   1:  PR[GP1:91,2] = PR[GP1:90,2] + 0.302;
   1:L PR[91] 10mm/sec CNT100;
   1:  PR[GP1:91,1] = PR[GP1:90,1] + 73.416;
   1:  PR[GP1:91,2] = PR[GP1:90,2] + 5.594;
   1:L PR[91] 10mm/sec CNT100;
   1:  PR[GP1:91,1] = PR[GP1:90,1] + 72.687;
   1:  PR[GP1:91,2] = PR[GP1:90,2] + 9.406;
   1:L PR[91] 10mm/sec CNT100;
   1:  PR[GP1:91,1] = PR[GP1:90,1] + 70.980;
   1:  PR[GP1:91,2] = PR[GP1:90,2] + 14.355;
   1:L PR[91] 10mm/sec CNT100;
   1:  PR[GP1:91,1] = PR[GP1:90,1] + 68.206;
   1:  PR[GP1:91,2] = PR[GP1:90,2] + 18.843;
   1:L PR[91] 10mm/sec CNT100;
   1:  PR[GP1:91,1] = PR[GP1:90,1] + 66.056;
   1:  PR[GP1:91,2] = PR[GP1:90,2] + 22.237;
   1:L PR[91] 10mm/sec CNT100;
   1:  PR[GP1:91,1] = PR[GP1:90,1] + 62.477;
   1:  PR[GP1:91,2] = PR[GP1:90,2] + 25.890;
   1:L PR[91] 10mm/sec CNT100;
   1:  PR[GP1:91,1] = PR[GP1:90,1] + 58.115;
   1:  PR[GP1:91,2] = PR[GP1:90,2] + 28.712;
   1:L PR[91] 10mm/sec CNT100;
   1:  PR[GP1:91,1] = PR[GP1:90,1] + 54.751;
   1:  PR[GP1:91,2] = PR[GP1:90,2] + 31.172;
   1:L PR[91] 10mm/sec CNT100;
   1:  PR[GP1:91,1] = PR[GP1:90,1] + 50.096;
   1:  PR[GP1:91,2] = PR[GP1:90,2] + 32.886;
   1:L PR[91] 10mm/sec CNT100;
   1:  PR[GP1:91,1] = PR[GP1:90,1] + 45.611;
   1:  PR[GP1:91,2] = PR[GP1:90,2] + 34.049;
   1:L PR[91] 10mm/sec CNT100;
   1:  PR[GP1:91,1] = PR[GP1:90,1] + 40.919;
   1:  PR[GP1:91,2] = PR[GP1:90,2] + 34.669;
   1:L PR[91] 10mm/sec CNT100;
   1:  PR[GP1:91,1] = PR[GP1:90,1] + 36.178;
   1:  PR[GP1:91,2] = PR[GP1:90,2] + 34.240;
   1:L PR[91] 10mm/sec CNT100;
   1:  PR[GP1:91,1] = PR[GP1:90,1] + 31.221;
   1:  PR[GP1:91,2] = PR[GP1:90,2] + 33.641;
   1:L PR[91] 10mm/sec CNT100;
   1:  PR[GP1:91,1] = PR[GP1:90,1] + 27.016;
   1:  PR[GP1:91,2] = PR[GP1:90,2] + 32.287;
   1:L PR[91] 10mm/sec CNT100;
   1:  PR[GP1:91,1] = PR[GP1:90,1] + 23.151;
   1:  PR[GP1:91,2] = PR[GP1:90,2] + 30.007;
   1:L PR[91] 10mm/sec CNT100;
   1:  PR[GP1:91,1] = PR[GP1:90,1] + 18.388;
   1:  PR[GP1:91,2] = PR[GP1:90,2] + 27.451;
   1:L PR[91] 10mm/sec CNT100;
   1:  PR[GP1:91,1] = PR[GP1:90,1] + 15.391;
   1:  PR[GP1:91,2] = PR[GP1:90,2] + 24.634;
   1:L PR[91] 10mm/sec CNT100;
   1:  PR[GP1:91,1] = PR[GP1:90,1] + 11.444;
   1:  PR[GP1:91,2] = PR[GP1:90,2] + 19.952;
   1:L PR[91] 10mm/sec CNT100;
   1:  PR[GP1:91,1] = PR[GP1:90,1] + 9.285;
   1:  PR[GP1:91,2] = PR[GP1:90,2] + 16.760;
   1:L PR[91] 10mm/sec CNT100;
   1:  PR[GP1:91,1] = PR[GP1:90,1] + 7.872;
   1:  PR[GP1:91,2] = PR[GP1:90,2] + 13.156;
   1:L PR[91] 10mm/sec CNT100;
   1:  PR[GP1:91,1] = PR[GP1:90,1] + 5.812;
   1:  PR[GP1:91,2] = PR[GP1:90,2] + 7.089;
   1:L PR[91] 10mm/sec CNT100;
   1:  PR[GP1:91,1] = PR[GP1:90,1] + 5.265;
   1:  PR[GP1:91,2] = PR[GP1:90,2] + 3.511;
   1:L PR[91] 10mm/sec CNT100;
   1:  PR[GP1:91,1] = PR[GP1:90,1] + 5.491;
   1:  PR[GP1:91,2] = PR[GP1:90,2] + 2.717;
   1:L PR[91] 10mm/sec CNT100;
   1:  PR[GP1:91,1] = PR[GP1:90,1] + -5.747;
   1:L PR[91] 10mm/sec CNT100;
   1:  PR[GP1:91,1] = PR[GP1:90,1] + -6.339;
   1:  PR[GP1:91,2] = PR[GP1:90,2] + 7.082;
   1:L PR[91] 10mm/sec CNT100;
   1:  PR[GP1:91,1] = PR[GP1:90,1] + -7.706;
   1:  PR[GP1:91,2] = PR[GP1:90,2] + 10.570;
   1:L PR[91] 10mm/sec CNT100;
   1:  PR[GP1:91,1] = PR[GP1:90,1] + -9.820;
   1:  PR[GP1:91,2] = PR[GP1:90,2] + 16.776;
   1:L PR[91] 10mm/sec CNT100;
   1:  PR[GP1:91,1] = PR[GP1:90,1] + -11.972;
   1:  PR[GP1:91,2] = PR[GP1:90,2] + 19.956;
   1:L PR[91] 10mm/sec CNT100;
   1:  PR[GP1:91,1] = PR[GP1:90,1] + -15.920;
   1:  PR[GP1:91,2] = PR[GP1:90,2] + 24.636;
   1:L PR[91] 10mm/sec CNT100;
   1:  PR[GP1:91,1] = PR[GP1:90,1] + -18.925;
   1:  PR[GP1:91,2] = PR[GP1:90,2] + 27.461;
   1:L PR[91] 10mm/sec CNT100;
   1:  PR[GP1:91,1] = PR[GP1:90,1] + -22.498;
   1:  PR[GP1:91,2] = PR[GP1:90,2] + 29.569;
   1:L PR[91] 10mm/sec CNT100;
   1:  PR[GP1:91,1] = PR[GP1:90,1] + -27.533;
   1:  PR[GP1:91,2] = PR[GP1:90,2] + 32.284;
   1:L PR[91] 10mm/sec CNT100;
   1:  PR[GP1:91,1] = PR[GP1:90,1] + -31.740;
   1:  PR[GP1:91,2] = PR[GP1:90,2] + 33.639;
   1:L PR[91] 10mm/sec CNT100;
   1:  PR[GP1:91,1] = PR[GP1:90,1] + -36.206;
   1:  PR[GP1:91,2] = PR[GP1:90,2] + 34.043;
   1:L PR[91] 10mm/sec CNT100;
   1:  PR[GP1:91,1] = PR[GP1:90,1] + -41.456;
   1:  PR[GP1:91,2] = PR[GP1:90,2] + 34.668;
   1:L PR[91] 10mm/sec CNT100;
   1:  PR[GP1:91,1] = PR[GP1:90,1] + -46.139;
   1:  PR[GP1:91,2] = PR[GP1:90,2] + 34.049;
   1:L PR[91] 10mm/sec CNT100;
   1:  PR[GP1:91,1] = PR[GP1:90,1] + -50.623;
   1:  PR[GP1:91,2] = PR[GP1:90,2] + 32.886;
   1:L PR[91] 10mm/sec CNT100;
   1:  PR[GP1:91,1] = PR[GP1:90,1] + -55.294;
   1:  PR[GP1:91,2] = PR[GP1:90,2] + 31.166;
   1:L PR[91] 10mm/sec CNT100;
   1:  PR[GP1:91,1] = PR[GP1:90,1] + -59.485;
   1:  PR[GP1:91,2] = PR[GP1:90,2] + 28.455;
   1:L PR[91] 10mm/sec CNT100;
   1:  PR[GP1:91,1] = PR[GP1:90,1] + -62.992;
   1:  PR[GP1:91,2] = PR[GP1:90,2] + 25.902;
   1:L PR[91] 10mm/sec CNT100;
   1:  PR[GP1:91,1] = PR[GP1:90,1] + -66.580;
   1:  PR[GP1:91,2] = PR[GP1:90,2] + 22.239;
   1:L PR[91] 10mm/sec CNT100;
   1:  PR[GP1:91,1] = PR[GP1:90,1] + -69.304;
   1:  PR[GP1:91,2] = PR[GP1:90,2] + 17.832;
   1:L PR[91] 10mm/sec CNT100;
   1:  PR[GP1:91,1] = PR[GP1:90,1] + -71.508;
   1:  PR[GP1:91,2] = PR[GP1:90,2] + 14.351;
   1:L PR[91] 10mm/sec CNT100;
   1:  PR[GP1:91,1] = PR[GP1:90,1] + -73.206;
   1:  PR[GP1:91,2] = PR[GP1:90,2] + 9.427;
   1:L PR[91] 10mm/sec CNT100;
   1:  PR[GP1:91,1] = PR[GP1:90,1] + -73.792;
   1:  PR[GP1:91,2] = PR[GP1:90,2] + 4.158;
   1:L PR[91] 10mm/sec CNT100;
   1:  PR[GP1:91,1] = PR[GP1:90,1] + -74.531;
   1:  PR[GP1:91,2] = PR[GP1:90,2] + 0.256;
   1:L PR[91] 10mm/sec CNT100;
   1:  PR[GP1:91,1] = PR[GP1:90,1] + -73.943;
   1:  PR[GP1:91,2] = PR[GP1:90,2] + -5.036;
   1:L PR[91] 10mm/sec CNT100;
   1:  PR[GP1:91,1] = PR[GP1:90,1] + -73.214;
   1:  PR[GP1:91,2] = PR[GP1:90,2] + -8.847;
   1:L PR[91] 10mm/sec CNT100;
   1:  PR[GP1:91,1] = PR[GP1:90,1] + -71.506;
   1:  PR[GP1:91,2] = PR[GP1:90,2] + -13.796;
   1:L PR[91] 10mm/sec CNT100;
   1:  PR[GP1:91,1] = PR[GP1:90,1] + -68.733;
   1:  PR[GP1:91,2] = PR[GP1:90,2] + -18.284;
   1:L PR[91] 10mm/sec CNT100;
   1:  PR[GP1:91,1] = PR[GP1:90,1] + -66.582;
   1:  PR[GP1:91,2] = PR[GP1:90,2] + -21.678;
   1:L PR[91] 10mm/sec CNT100;
   1:  PR[GP1:91,1] = PR[GP1:90,1] + -63.003;
   1:  PR[GP1:91,2] = PR[GP1:90,2] + -25.332;
   1:L PR[91] 10mm/sec CNT100;
   1:  PR[GP1:91,1] = PR[GP1:90,1] + -58.642;
   1:  PR[GP1:91,2] = PR[GP1:90,2] + -28.154;
   1:L PR[91] 10mm/sec CNT100;
   1:  PR[GP1:91,1] = PR[GP1:90,1] + -55.278;
   1:  PR[GP1:91,2] = PR[GP1:90,2] + -30.614;
   1:L PR[91] 10mm/sec CNT100;
   1:  PR[GP1:91,1] = PR[GP1:90,1] + -50.623;
   1:  PR[GP1:91,2] = PR[GP1:90,2] + -32.328;
   1:L PR[91] 10mm/sec CNT100;
   1:  PR[GP1:91,1] = PR[GP1:90,1] + -46.139;
   1:  PR[GP1:91,2] = PR[GP1:90,2] + -33.491;
   1:L PR[91] 10mm/sec CNT100;
   1:  PR[GP1:91,1] = PR[GP1:90,1] + -41.447;
   1:  PR[GP1:91,2] = PR[GP1:90,2] + -34.111;
   1:L PR[91] 10mm/sec CNT100;
   1:  PR[GP1:91,1] = PR[GP1:90,1] + -36.706;
   1:  PR[GP1:91,2] = PR[GP1:90,2] + -33.682;
   1:L PR[91] 10mm/sec CNT100;
   1:  PR[GP1:91,1] = PR[GP1:90,1] + -31.749;
   1:  PR[GP1:91,2] = PR[GP1:90,2] + -33.084;
   1:L PR[91] 10mm/sec CNT100;
   1:  PR[GP1:91,1] = PR[GP1:90,1] + -27.544;
   1:  PR[GP1:91,2] = PR[GP1:90,2] + -31.730;
   1:L PR[91] 10mm/sec CNT100;
   1:  PR[GP1:91,1] = PR[GP1:90,1] + -23.679;
   1:  PR[GP1:91,2] = PR[GP1:90,2] + -29.449;
   1:L PR[91] 10mm/sec CNT100;
   1:  PR[GP1:91,1] = PR[GP1:90,1] + -18.916;
   1:  PR[GP1:91,2] = PR[GP1:90,2] + -26.894;
   1:L PR[91] 10mm/sec CNT100;
   1:  PR[GP1:91,1] = PR[GP1:90,1] + -15.920;
   1:  PR[GP1:91,2] = PR[GP1:90,2] + -24.078;
   1:L PR[91] 10mm/sec CNT100;
   1:  PR[GP1:91,1] = PR[GP1:90,1] + -11.972;
   1:  PR[GP1:91,2] = PR[GP1:90,2] + -19.398;
   1:L PR[91] 10mm/sec CNT100;
   1:  PR[GP1:91,1] = PR[GP1:90,1] + -9.813;
   1:  PR[GP1:91,2] = PR[GP1:90,2] + -16.206;
   1:L PR[91] 10mm/sec CNT100;
   1:  PR[GP1:91,1] = PR[GP1:90,1] + -8.401;
   1:  PR[GP1:91,2] = PR[GP1:90,2] + -12.602;
   1:L PR[91] 10mm/sec CNT100;
   1:  PR[GP1:91,1] = PR[GP1:90,1] + -6.339;
   1:  PR[GP1:91,2] = PR[GP1:90,2] + -6.530;
   1:L PR[91] 10mm/sec CNT100;
   1:  PR[GP1:91,1] = PR[GP1:90,1] + -5.791;
   1:  PR[GP1:91,2] = PR[GP1:90,2] + -2.953;
   1:L PR[91] 10mm/sec CNT100;
   1:  PR[GP1:91,1] = PR[GP1:90,1] + -6.017;
   1:  PR[GP1:91,2] = PR[GP1:90,2] + -2.159;
   1:L PR[91] 10mm/sec CNT100;
   1:  PR[GP1:91,1] = PR[GP1:90,1] + 5.220;
   1:L PR[91] 10mm/sec CNT100;
   1:  PR[GP1:91,1] = PR[GP1:90,1] + 5.692;
   1:  PR[GP1:91,2] = PR[GP1:90,2] + -6.161;
   1:  PR[GP1:91,3] = PR[GP1:90,3] + 12.505;
   1:L PR[91] 10mm/sec CNT100;
   1:  PR[GP1:91,1] = PR[GP1:90,1] + 6.815;
   1:  PR[GP1:91,2] = PR[GP1:90,2] + -9.028;
   1:L PR[91] 10mm/sec CNT100;
   1:  PR[GP1:91,1] = PR[GP1:90,1] + 9.291;
   1:  PR[GP1:91,2] = PR[GP1:90,2] + -16.294;
   1:L PR[91] 10mm/sec CNT100;
   1:  PR[GP1:91,1] = PR[GP1:90,1] + 11.082;
   1:  PR[GP1:91,2] = PR[GP1:90,2] + -18.941;
   1:L PR[91] 10mm/sec CNT100;
   1:  PR[GP1:91,1] = PR[GP1:90,1] + 15.708;
   1:  PR[GP1:91,2] = PR[GP1:90,2] + -24.429;
   1:L PR[91] 10mm/sec CNT100;
   1:  PR[GP1:91,1] = PR[GP1:90,1] + 18.278;
   1:  PR[GP1:91,2] = PR[GP1:90,2] + -26.845;
   1:L PR[91] 10mm/sec CNT100;
   1:  PR[GP1:91,1] = PR[GP1:90,1] + 21.337;
   1:  PR[GP1:91,2] = PR[GP1:90,2] + -28.650;
   1:L PR[91] 10mm/sec CNT100;
   1:  PR[GP1:91,1] = PR[GP1:90,1] + 27.239;
   1:  PR[GP1:91,2] = PR[GP1:90,2] + -31.833;
   1:L PR[91] 10mm/sec CNT100;
   1:  PR[GP1:91,1] = PR[GP1:90,1] + 30.929;
   1:  PR[GP1:91,2] = PR[GP1:90,2] + -33.022;
   1:L PR[91] 10mm/sec CNT100;
   1:  PR[GP1:91,1] = PR[GP1:90,1] + 34.855;
   1:  PR[GP1:91,2] = PR[GP1:90,2] + -33.376;
   1:L PR[91] 10mm/sec CNT100;
   1:  PR[GP1:91,1] = PR[GP1:90,1] + 41.008;
   1:  PR[GP1:91,2] = PR[GP1:90,2] + -34.110;
   1:L PR[91] 10mm/sec CNT100;
   1:  PR[GP1:91,1] = PR[GP1:90,1] + 45.203;
   1:  PR[GP1:91,2] = PR[GP1:90,2] + -33.556;
   1:L PR[91] 10mm/sec CNT100;
   1:  PR[GP1:91,1] = PR[GP1:90,1] + 50.461;
   1:  PR[GP1:91,2] = PR[GP1:90,2] + -32.192;
   1:L PR[91] 10mm/sec CNT100;
   1:  PR[GP1:91,1] = PR[GP1:90,1] + 54.708;
   1:  PR[GP1:91,2] = PR[GP1:90,2] + -30.629;
   1:L PR[91] 10mm/sec CNT100;
   1:  PR[GP1:91,1] = PR[GP1:90,1] + 58.519;
   1:  PR[GP1:91,2] = PR[GP1:90,2] + -28.163;
   1:L PR[91] 10mm/sec CNT100;
   1:  PR[GP1:91,1] = PR[GP1:90,1] + 62.631;
   1:  PR[GP1:91,2] = PR[GP1:90,2] + -25.170;
   1:L PR[91] 10mm/sec CNT100;
   1:  PR[GP1:91,1] = PR[GP1:90,1] + 65.923;
   1:  PR[GP1:91,2] = PR[GP1:90,2] + -21.809;
   1:L PR[91] 10mm/sec CNT100;
   1:  PR[GP1:91,1] = PR[GP1:90,1] + 68.425;
   1:  PR[GP1:91,2] = PR[GP1:90,2] + -17.762;
   1:L PR[91] 10mm/sec CNT100;
   1:  PR[GP1:91,1] = PR[GP1:90,1] + 71.009;
   1:  PR[GP1:91,2] = PR[GP1:90,2] + -13.681;
   1:L PR[91] 10mm/sec CNT100;
   1:  PR[GP1:91,1] = PR[GP1:90,1] + 72.575;
   1:  PR[GP1:91,2] = PR[GP1:90,2] + -9.141;
   1:L PR[91] 10mm/sec CNT100;
   1:  PR[GP1:91,1] = PR[GP1:90,1] + 73.116;
   1:  PR[GP1:91,2] = PR[GP1:90,2] + -4.276;
   1:L PR[91] 10mm/sec CNT100;
   1:  PR[GP1:91,1] = PR[GP1:90,1] + 73.983;
   1:  PR[GP1:91,2] = PR[GP1:90,2] + 0.302;
   1:L PR[91] 10mm/sec CNT100;
   1:  PR[GP1:91,1] = PR[GP1:90,1] + 73.438;
   1:  PR[GP1:91,2] = PR[GP1:90,2] + 5.206;
   1:L PR[91] 10mm/sec CNT100;
   1:  PR[GP1:91,1] = PR[GP1:90,1] + 72.583;
   1:  PR[GP1:91,2] = PR[GP1:90,2] + 9.677;
   1:L PR[91] 10mm/sec CNT100;
   1:  PR[GP1:91,1] = PR[GP1:90,1] + 71.008;
   1:  PR[GP1:91,2] = PR[GP1:90,2] + 14.242;
   1:L PR[91] 10mm/sec CNT100;
   1:  PR[GP1:91,1] = PR[GP1:90,1] + 68.448;
   1:  PR[GP1:91,2] = PR[GP1:90,2] + 18.385;
   1:L PR[91] 10mm/sec CNT100;
   1:  PR[GP1:91,1] = PR[GP1:90,1] + 65.926;
   1:  PR[GP1:91,2] = PR[GP1:90,2] + 22.365;
   1:L PR[91] 10mm/sec CNT100;
   1:  PR[GP1:91,1] = PR[GP1:90,1] + 62.643;
   1:  PR[GP1:91,2] = PR[GP1:90,2] + 25.716;
   1:L PR[91] 10mm/sec CNT100;
   1:  PR[GP1:91,1] = PR[GP1:90,1] + 58.637;
   1:  PR[GP1:91,2] = PR[GP1:90,2] + 28.308;
   1:L PR[91] 10mm/sec CNT100;
   1:  PR[GP1:91,1] = PR[GP1:90,1] + 54.692;
   1:  PR[GP1:91,2] = PR[GP1:90,2] + 31.193;
   1:L PR[91] 10mm/sec CNT100;
   1:  PR[GP1:91,1] = PR[GP1:90,1] + 50.461;
   1:  PR[GP1:91,2] = PR[GP1:90,2] + 32.750;
   1:L PR[91] 10mm/sec CNT100;
   1:  PR[GP1:91,1] = PR[GP1:90,1] + 45.203;
   1:  PR[GP1:91,2] = PR[GP1:90,2] + 34.114;
   1:L PR[91] 10mm/sec CNT100;
   1:  PR[GP1:91,1] = PR[GP1:90,1] + 41.000;
   1:  PR[GP1:91,2] = PR[GP1:90,2] + 34.669;
   1:L PR[91] 10mm/sec CNT100;
   1:  PR[GP1:91,1] = PR[GP1:90,1] + 36.749;
   1:  PR[GP1:91,2] = PR[GP1:90,2] + 34.285;
   1:L PR[91] 10mm/sec CNT100;
   1:  PR[GP1:91,1] = PR[GP1:90,1] + 30.938;
   1:  PR[GP1:91,2] = PR[GP1:90,2] + 33.582;
   1:L PR[91] 10mm/sec CNT100;
   1:  PR[GP1:91,1] = PR[GP1:90,1] + 27.250;
   1:  PR[GP1:91,2] = PR[GP1:90,2] + 32.395;
   1:L PR[91] 10mm/sec CNT100;
   1:  PR[GP1:91,1] = PR[GP1:90,1] + 23.852;
   1:  PR[GP1:91,2] = PR[GP1:90,2] + 30.390;
   1:L PR[91] 10mm/sec CNT100;
   1:  PR[GP1:91,1] = PR[GP1:90,1] + 18.269;
   1:  PR[GP1:91,2] = PR[GP1:90,2] + 27.395;
   1:L PR[91] 10mm/sec CNT100;
   1:  PR[GP1:91,1] = PR[GP1:90,1] + 15.708;
   1:  PR[GP1:91,2] = PR[GP1:90,2] + 24.986;
   1:L PR[91] 10mm/sec CNT100;
   1:  PR[GP1:91,1] = PR[GP1:90,1] + 11.082;
   1:  PR[GP1:91,2] = PR[GP1:90,2] + 19.499;
   1:L PR[91] 10mm/sec CNT100;
   1:  PR[GP1:91,1] = PR[GP1:90,1] + 9.283;
   1:  PR[GP1:91,2] = PR[GP1:90,2] + 16.840;
   1:L PR[91] 10mm/sec CNT100;
   1:  PR[GP1:91,1] = PR[GP1:90,1] + 8.106;
   1:  PR[GP1:91,2] = PR[GP1:90,2] + 13.834;
   1:L PR[91] 10mm/sec CNT100;
   1:  PR[GP1:91,1] = PR[GP1:90,1] + 5.692;
   1:  PR[GP1:91,2] = PR[GP1:90,2] + 6.726;
   1:L PR[91] 10mm/sec CNT100;
   1:  PR[GP1:91,1] = PR[GP1:90,1] + 5.245;
   1:  PR[GP1:91,2] = PR[GP1:90,2] + 3.808;
   1:L PR[91] 10mm/sec CNT100;
   1:  PR[GP1:91,1] = PR[GP1:90,1] + 5.463;
   1:  PR[GP1:91,2] = PR[GP1:90,2] + 3.042;
   1:L PR[91] 10mm/sec CNT100;
   1:  PR[GP1:91,1] = PR[GP1:90,1] + -5.719;
   1:L PR[91] 10mm/sec CNT100;
   1:  PR[GP1:91,1] = PR[GP1:90,1] + -6.218;
   1:  PR[GP1:91,2] = PR[GP1:90,2] + 6.719;
   1:L PR[91] 10mm/sec CNT100;
   1:  PR[GP1:91,1] = PR[GP1:90,1] + -7.341;
   1:  PR[GP1:91,2] = PR[GP1:90,2] + 9.586;
   1:L PR[91] 10mm/sec CNT100;
   1:  PR[GP1:91,1] = PR[GP1:90,1] + -9.819;
   1:  PR[GP1:91,2] = PR[GP1:90,2] + 16.857;
   1:L PR[91] 10mm/sec CNT100;
   1:  PR[GP1:91,1] = PR[GP1:90,1] + -11.611;
   1:  PR[GP1:91,2] = PR[GP1:90,2] + 19.505;
   1:L PR[91] 10mm/sec CNT100;
   1:  PR[GP1:91,1] = PR[GP1:90,1] + -16.236;
   1:  PR[GP1:91,2] = PR[GP1:90,2] + 24.988;
   1:L PR[91] 10mm/sec CNT100;
   1:  PR[GP1:91,1] = PR[GP1:90,1] + -18.807;
   1:  PR[GP1:91,2] = PR[GP1:90,2] + 27.405;
   1:L PR[91] 10mm/sec CNT100;
   1:  PR[GP1:91,1] = PR[GP1:90,1] + -21.866;
   1:  PR[GP1:91,2] = PR[GP1:90,2] + 29.210;
   1:L PR[91] 10mm/sec CNT100;
   1:  PR[GP1:91,1] = PR[GP1:90,1] + -27.767;
   1:  PR[GP1:91,2] = PR[GP1:90,2] + 32.392;
   1:L PR[91] 10mm/sec CNT100;
   1:  PR[GP1:91,1] = PR[GP1:90,1] + -31.458;
   1:  PR[GP1:91,2] = PR[GP1:90,2] + 33.581;
   1:L PR[91] 10mm/sec CNT100;
   1:  PR[GP1:91,1] = PR[GP1:90,1] + -35.384;
   1:  PR[GP1:91,2] = PR[GP1:90,2] + 33.935;
   1:L PR[91] 10mm/sec CNT100;
   1:  PR[GP1:91,1] = PR[GP1:90,1] + -41.537;
   1:  PR[GP1:91,2] = PR[GP1:90,2] + 34.668;
   1:L PR[91] 10mm/sec CNT100;
   1:  PR[GP1:91,1] = PR[GP1:90,1] + -45.731;
   1:  PR[GP1:91,2] = PR[GP1:90,2] + 34.114;
   1:L PR[91] 10mm/sec CNT100;
   1:  PR[GP1:91,1] = PR[GP1:90,1] + -50.988;
   1:  PR[GP1:91,2] = PR[GP1:90,2] + 32.750;
   1:L PR[91] 10mm/sec CNT100;
   1:  PR[GP1:91,1] = PR[GP1:90,1] + -55.235;
   1:  PR[GP1:91,2] = PR[GP1:90,2] + 31.186;
   1:L PR[91] 10mm/sec CNT100;
   1:  PR[GP1:91,1] = PR[GP1:90,1] + -59.046;
   1:  PR[GP1:91,2] = PR[GP1:90,2] + 28.721;
   1:L PR[91] 10mm/sec CNT100;
   1:  PR[GP1:91,1] = PR[GP1:90,1] + -63.158;
   1:  PR[GP1:91,2] = PR[GP1:90,2] + 25.727;
   1:L PR[91] 10mm/sec CNT100;
   1:  PR[GP1:91,1] = PR[GP1:90,1] + -66.450;
   1:  PR[GP1:91,2] = PR[GP1:90,2] + 22.367;
   1:L PR[91] 10mm/sec CNT100;
   1:  PR[GP1:91,1] = PR[GP1:90,1] + -68.952;
   1:  PR[GP1:91,2] = PR[GP1:90,2] + 18.320;
   1:L PR[91] 10mm/sec CNT100;
   1:  PR[GP1:91,1] = PR[GP1:90,1] + -71.536;
   1:  PR[GP1:91,2] = PR[GP1:90,2] + 14.238;
   1:L PR[91] 10mm/sec CNT100;
   1:  PR[GP1:91,1] = PR[GP1:90,1] + -73.102;
   1:  PR[GP1:91,2] = PR[GP1:90,2] + 9.698;
   1:L PR[91] 10mm/sec CNT100;
   1:  PR[GP1:91,1] = PR[GP1:90,1] + -73.643;
   1:  PR[GP1:91,2] = PR[GP1:90,2] + 4.832;
   1:L PR[91] 10mm/sec CNT100;
   1:  PR[GP1:91,1] = PR[GP1:90,1] + -74.510;
   1:  PR[GP1:91,2] = PR[GP1:90,2] + 0.256;
   1:L PR[91] 10mm/sec CNT100;
   1:  PR[GP1:91,1] = PR[GP1:90,1] + -73.965;
   1:  PR[GP1:91,2] = PR[GP1:90,2] + -4.648;
   1:L PR[91] 10mm/sec CNT100;
   1:  PR[GP1:91,1] = PR[GP1:90,1] + -73.110;
   1:  PR[GP1:91,2] = PR[GP1:90,2] + -9.118;
   1:L PR[91] 10mm/sec CNT100;
   1:  PR[GP1:91,1] = PR[GP1:90,1] + -71.535;
   1:  PR[GP1:91,2] = PR[GP1:90,2] + -13.683;
   1:L PR[91] 10mm/sec CNT100;
   1:  PR[GP1:91,1] = PR[GP1:90,1] + -68.974;
   1:  PR[GP1:91,2] = PR[GP1:90,2] + -17.825;
   1:L PR[91] 10mm/sec CNT100;
   1:  PR[GP1:91,1] = PR[GP1:90,1] + -66.453;
   1:  PR[GP1:91,2] = PR[GP1:90,2] + -21.806;
   1:L PR[91] 10mm/sec CNT100;
   1:  PR[GP1:91,1] = PR[GP1:90,1] + -63.170;
   1:  PR[GP1:91,2] = PR[GP1:90,2] + -25.157;
   1:L PR[91] 10mm/sec CNT100;
   1:  PR[GP1:91,1] = PR[GP1:90,1] + -59.163;
   1:  PR[GP1:91,2] = PR[GP1:90,2] + -27.750;
   1:L PR[91] 10mm/sec CNT100;
   1:  PR[GP1:91,1] = PR[GP1:90,1] + -55.219;
   1:  PR[GP1:91,2] = PR[GP1:90,2] + -30.634;
   1:L PR[91] 10mm/sec CNT100;
   1:  PR[GP1:91,1] = PR[GP1:90,1] + -50.988;
   1:  PR[GP1:91,2] = PR[GP1:90,2] + -32.192;
   1:L PR[91] 10mm/sec CNT100;
   1:  PR[GP1:91,1] = PR[GP1:90,1] + -45.731;
   1:  PR[GP1:91,2] = PR[GP1:90,2] + -33.556;
   1:L PR[91] 10mm/sec CNT100;
   1:  PR[GP1:91,1] = PR[GP1:90,1] + -41.528;
   1:  PR[GP1:91,2] = PR[GP1:90,2] + -34.111;
   1:L PR[91] 10mm/sec CNT100;
   1:  PR[GP1:91,1] = PR[GP1:90,1] + -37.278;
   1:  PR[GP1:91,2] = PR[GP1:90,2] + -33.727;
   1:L PR[91] 10mm/sec CNT100;
   1:  PR[GP1:91,1] = PR[GP1:90,1] + -31.467;
   1:  PR[GP1:91,2] = PR[GP1:90,2] + -33.025;
   1:L PR[91] 10mm/sec CNT100;
   1:  PR[GP1:91,1] = PR[GP1:90,1] + -27.778;
   1:  PR[GP1:91,2] = PR[GP1:90,2] + -31.837;
   1:L PR[91] 10mm/sec CNT100;
   1:  PR[GP1:91,1] = PR[GP1:90,1] + -24.381;
   1:  PR[GP1:91,2] = PR[GP1:90,2] + -29.833;
   1:L PR[91] 10mm/sec CNT100;
   1:  PR[GP1:91,1] = PR[GP1:90,1] + -18.798;
   1:  PR[GP1:91,2] = PR[GP1:90,2] + -26.838;
   1:L PR[91] 10mm/sec CNT100;
   1:  PR[GP1:91,1] = PR[GP1:90,1] + -16.236;
   1:  PR[GP1:91,2] = PR[GP1:90,2] + -24.430;
   1:L PR[91] 10mm/sec CNT100;
   1:  PR[GP1:91,1] = PR[GP1:90,1] + -11.611;
   1:  PR[GP1:91,2] = PR[GP1:90,2] + -18.946;
   1:L PR[91] 10mm/sec CNT100;
   1:  PR[GP1:91,1] = PR[GP1:90,1] + -9.812;
   1:  PR[GP1:91,2] = PR[GP1:90,2] + -16.287;
   1:L PR[91] 10mm/sec CNT100;
   1:  PR[GP1:91,1] = PR[GP1:90,1] + -8.634;
   1:  PR[GP1:91,2] = PR[GP1:90,2] + -13.281;
   1:L PR[91] 10mm/sec CNT100;
   1:  PR[GP1:91,1] = PR[GP1:90,1] + -6.218;
   1:  PR[GP1:91,2] = PR[GP1:90,2] + -6.167;
   1:L PR[91] 10mm/sec CNT100;
   1:  PR[GP1:91,1] = PR[GP1:90,1] + -5.772;
   1:  PR[GP1:91,2] = PR[GP1:90,2] + -3.250;
   1:L PR[91] 10mm/sec CNT100;
   1:  PR[GP1:91,1] = PR[GP1:90,1] + -5.990;
   1:  PR[GP1:91,2] = PR[GP1:90,2] + -2.483;
   1:L PR[91] 10mm/sec CNT100;
   1:  PR[GP1:91,1] = PR[GP1:90,1] + 5.193;
   1:L PR[91] 10mm/sec CNT100;
   1:  PR[GP1:91,1] = PR[GP1:90,1] + 5.571;
   1:  PR[GP1:91,2] = PR[GP1:90,2] + -5.799;
   1:  PR[GP1:91,3] = PR[GP1:90,3] + 13.115;
   1:L PR[91] 10mm/sec CNT100;
   1:  PR[GP1:91,1] = PR[GP1:90,1] + 6.451;
   1:  PR[GP1:91,2] = PR[GP1:90,2] + -8.044;
   1:L PR[91] 10mm/sec CNT100;
   1:  PR[GP1:91,1] = PR[GP1:90,1] + 9.289;
   1:  PR[GP1:91,2] = PR[GP1:90,2] + -16.374;
   1:L PR[91] 10mm/sec CNT100;
   1:  PR[GP1:91,1] = PR[GP1:90,1] + 10.721;
   1:  PR[GP1:91,2] = PR[GP1:90,2] + -18.489;
   1:L PR[91] 10mm/sec CNT100;
   1:  PR[GP1:91,1] = PR[GP1:90,1] + 16.024;
   1:  PR[GP1:91,2] = PR[GP1:90,2] + -24.781;
   1:L PR[91] 10mm/sec CNT100;
   1:  PR[GP1:91,1] = PR[GP1:90,1] + 18.160;
   1:  PR[GP1:91,2] = PR[GP1:90,2] + -26.789;
   1:L PR[91] 10mm/sec CNT100;
   1:  PR[GP1:91,1] = PR[GP1:90,1] + 20.706;
   1:  PR[GP1:91,2] = PR[GP1:90,2] + -28.291;
   1:L PR[91] 10mm/sec CNT100;
   1:  PR[GP1:91,1] = PR[GP1:90,1] + 27.473;
   1:  PR[GP1:91,2] = PR[GP1:90,2] + -31.941;
   1:L PR[91] 10mm/sec CNT100;
   1:  PR[GP1:91,1] = PR[GP1:90,1] + 30.647;
   1:  PR[GP1:91,2] = PR[GP1:90,2] + -32.963;
   1:L PR[91] 10mm/sec CNT100;
   1:  PR[GP1:91,1] = PR[GP1:90,1] + 34.032;
   1:  PR[GP1:91,2] = PR[GP1:90,2] + -33.269;
   1:L PR[91] 10mm/sec CNT100;
   1:  PR[GP1:91,1] = PR[GP1:90,1] + 41.089;
   1:  PR[GP1:91,2] = PR[GP1:90,2] + -34.110;
   1:L PR[91] 10mm/sec CNT100;
   1:  PR[GP1:91,1] = PR[GP1:90,1] + 44.795;
   1:  PR[GP1:91,2] = PR[GP1:90,2] + -33.620;
   1:L PR[91] 10mm/sec CNT100;
   1:  PR[GP1:91,1] = PR[GP1:90,1] + 50.826;
   1:  PR[GP1:91,2] = PR[GP1:90,2] + -32.057;
   1:L PR[91] 10mm/sec CNT100;
   1:  PR[GP1:91,1] = PR[GP1:90,1] + 54.649;
   1:  PR[GP1:91,2] = PR[GP1:90,2] + -30.649;
   1:L PR[91] 10mm/sec CNT100;
   1:  PR[GP1:91,1] = PR[GP1:90,1] + 58.080;
   1:  PR[GP1:91,2] = PR[GP1:90,2] + -28.429;
   1:L PR[91] 10mm/sec CNT100;
   1:  PR[GP1:91,1] = PR[GP1:90,1] + 62.798;
   1:  PR[GP1:91,2] = PR[GP1:90,2] + -24.995;
   1:L PR[91] 10mm/sec CNT100;
   1:  PR[GP1:91,1] = PR[GP1:90,1] + 65.794;
   1:  PR[GP1:91,2] = PR[GP1:90,2] + -21.937;
   1:L PR[91] 10mm/sec CNT100;
   1:  PR[GP1:91,1] = PR[GP1:90,1] + 68.073;
   1:  PR[GP1:91,2] = PR[GP1:90,2] + -18.250;
   1:L PR[91] 10mm/sec CNT100;
   1:  PR[GP1:91,1] = PR[GP1:90,1] + 71.037;
   1:  PR[GP1:91,2] = PR[GP1:90,2] + -13.568;
   1:L PR[91] 10mm/sec CNT100;
   1:  PR[GP1:91,1] = PR[GP1:90,1] + 72.471;
   1:  PR[GP1:91,2] = PR[GP1:90,2] + -9.412;
   1:L PR[91] 10mm/sec CNT100;
   1:  PR[GP1:91,1] = PR[GP1:90,1] + 72.967;
   1:  PR[GP1:91,2] = PR[GP1:90,2] + -4.950;
   1:L PR[91] 10mm/sec CNT100;
   1:  PR[GP1:91,1] = PR[GP1:90,1] + 73.962;
   1:  PR[GP1:91,2] = PR[GP1:90,2] + 0.302;
   1:L PR[91] 10mm/sec CNT100;
   1:  PR[GP1:91,1] = PR[GP1:90,1] + 73.460;
   1:  PR[GP1:91,2] = PR[GP1:90,2] + 4.818;
   1:L PR[91] 10mm/sec CNT100;
   1:  PR[GP1:91,1] = PR[GP1:90,1] + 72.479;
   1:  PR[GP1:91,2] = PR[GP1:90,2] + 9.948;
   1:L PR[91] 10mm/sec CNT100;
   1:  PR[GP1:91,1] = PR[GP1:90,1] + 71.036;
   1:  PR[GP1:91,2] = PR[GP1:90,2] + 14.129;
   1:L PR[91] 10mm/sec CNT100;
   1:  PR[GP1:91,1] = PR[GP1:90,1] + 68.690;
   1:  PR[GP1:91,2] = PR[GP1:90,2] + 17.926;
   1:L PR[91] 10mm/sec CNT100;
   1:  PR[GP1:91,1] = PR[GP1:90,1] + 65.796;
   1:  PR[GP1:91,2] = PR[GP1:90,2] + 22.493;
   1:L PR[91] 10mm/sec CNT100;
   1:  PR[GP1:91,1] = PR[GP1:90,1] + 62.809;
   1:  PR[GP1:91,2] = PR[GP1:90,2] + 25.542;
   1:L PR[91] 10mm/sec CNT100;
   1:  PR[GP1:91,1] = PR[GP1:90,1] + 59.158;
   1:  PR[GP1:91,2] = PR[GP1:90,2] + 27.904;
   1:L PR[91] 10mm/sec CNT100;
   1:  PR[GP1:91,1] = PR[GP1:90,1] + 54.632;
   1:  PR[GP1:91,2] = PR[GP1:90,2] + 31.213;
   1:L PR[91] 10mm/sec CNT100;
   1:  PR[GP1:91,1] = PR[GP1:90,1] + 50.826;
   1:  PR[GP1:91,2] = PR[GP1:90,2] + 32.615;
   1:L PR[91] 10mm/sec CNT100;
   1:  PR[GP1:91,1] = PR[GP1:90,1] + 44.795;
   1:  PR[GP1:91,2] = PR[GP1:90,2] + 34.178;
   1:L PR[91] 10mm/sec CNT100;
   1:  PR[GP1:91,1] = PR[GP1:90,1] + 41.080;
   1:  PR[GP1:91,2] = PR[GP1:90,2] + 34.669;
   1:L PR[91] 10mm/sec CNT100;
   1:  PR[GP1:91,1] = PR[GP1:90,1] + 37.320;
   1:  PR[GP1:91,2] = PR[GP1:90,2] + 34.329;
   1:L PR[91] 10mm/sec CNT100;
   1:  PR[GP1:91,1] = PR[GP1:90,1] + 30.656;
   1:  PR[GP1:91,2] = PR[GP1:90,2] + 33.524;
   1:L PR[91] 10mm/sec CNT100;
   1:  PR[GP1:91,1] = PR[GP1:90,1] + 27.484;
   1:  PR[GP1:91,2] = PR[GP1:90,2] + 32.502;
   1:L PR[91] 10mm/sec CNT100;
   1:  PR[GP1:91,1] = PR[GP1:90,1] + 24.553;
   1:  PR[GP1:91,2] = PR[GP1:90,2] + 30.773;
   1:L PR[91] 10mm/sec CNT100;
   1:  PR[GP1:91,1] = PR[GP1:90,1] + 18.151;
   1:  PR[GP1:91,2] = PR[GP1:90,2] + 27.338;
   1:L PR[91] 10mm/sec CNT100;
   1:  PR[GP1:91,1] = PR[GP1:90,1] + 16.024;
   1:  PR[GP1:91,2] = PR[GP1:90,2] + 25.339;
   1:L PR[91] 10mm/sec CNT100;
   1:  PR[GP1:91,1] = PR[GP1:90,1] + 10.721;
   1:  PR[GP1:91,2] = PR[GP1:90,2] + 19.047;
   1:L PR[91] 10mm/sec CNT100;
   1:  PR[GP1:91,1] = PR[GP1:90,1] + 9.282;
   1:  PR[GP1:91,2] = PR[GP1:90,2] + 16.921;
   1:L PR[91] 10mm/sec CNT100;
   1:  PR[GP1:91,1] = PR[GP1:90,1] + 8.339;
   1:  PR[GP1:91,2] = PR[GP1:90,2] + 14.513;
   1:L PR[91] 10mm/sec CNT100;
   1:  PR[GP1:91,1] = PR[GP1:90,1] + 5.571;
   1:  PR[GP1:91,2] = PR[GP1:90,2] + 6.363;
   1:L PR[91] 10mm/sec CNT100;
   1:  PR[GP1:91,1] = PR[GP1:90,1] + 5.225;
   1:  PR[GP1:91,2] = PR[GP1:90,2] + 4.106;
   1:L PR[91] 10mm/sec CNT100;
   1:  PR[GP1:91,1] = PR[GP1:90,1] + 5.436;
   1:  PR[GP1:91,2] = PR[GP1:90,2] + 3.367;
   1:L PR[91] 10mm/sec CNT100;
   1:  PR[GP1:91,1] = PR[GP1:90,1] + -5.692;
   1:L PR[91] 10mm/sec CNT100;
   1:  PR[GP1:91,1] = PR[GP1:90,1] + -6.098;
   1:  PR[GP1:91,2] = PR[GP1:90,2] + 6.357;
   1:L PR[91] 10mm/sec CNT100;
   1:  PR[GP1:91,1] = PR[GP1:90,1] + -6.977;
   1:  PR[GP1:91,2] = PR[GP1:90,2] + 8.601;
   1:L PR[91] 10mm/sec CNT100;
   1:  PR[GP1:91,1] = PR[GP1:90,1] + -9.818;
   1:  PR[GP1:91,2] = PR[GP1:90,2] + 16.938;
   1:L PR[91] 10mm/sec CNT100;
   1:  PR[GP1:91,1] = PR[GP1:90,1] + -11.249;
   1:  PR[GP1:91,2] = PR[GP1:90,2] + 19.053;
   1:L PR[91] 10mm/sec CNT100;
   1:  PR[GP1:91,1] = PR[GP1:90,1] + -16.553;
   1:  PR[GP1:91,2] = PR[GP1:90,2] + 25.340;
   1:L PR[91] 10mm/sec CNT100;
   1:  PR[GP1:91,1] = PR[GP1:90,1] + -18.690;
   1:  PR[GP1:91,2] = PR[GP1:90,2] + 27.349;
   1:L PR[91] 10mm/sec CNT100;
   1:  PR[GP1:91,1] = PR[GP1:90,1] + -21.235;
   1:  PR[GP1:91,2] = PR[GP1:90,2] + 28.851;
   1:L PR[91] 10mm/sec CNT100;
   1:  PR[GP1:91,1] = PR[GP1:90,1] + -28.002;
   1:  PR[GP1:91,2] = PR[GP1:90,2] + 32.500;
   1:L PR[91] 10mm/sec CNT100;
   1:  PR[GP1:91,1] = PR[GP1:90,1] + -31.176;
   1:  PR[GP1:91,2] = PR[GP1:90,2] + 33.522;
   1:L PR[91] 10mm/sec CNT100;
   1:  PR[GP1:91,1] = PR[GP1:90,1] + -34.561;
   1:  PR[GP1:91,2] = PR[GP1:90,2] + 33.828;
   1:L PR[91] 10mm/sec CNT100;
   1:  PR[GP1:91,1] = PR[GP1:90,1] + -41.617;
   1:  PR[GP1:91,2] = PR[GP1:90,2] + 34.668;
   1:L PR[91] 10mm/sec CNT100;
   1:  PR[GP1:91,1] = PR[GP1:90,1] + -45.324;
   1:  PR[GP1:91,2] = PR[GP1:90,2] + 34.178;
   1:L PR[91] 10mm/sec CNT100;
   1:  PR[GP1:91,1] = PR[GP1:90,1] + -51.354;
   1:  PR[GP1:91,2] = PR[GP1:90,2] + 32.614;
   1:L PR[91] 10mm/sec CNT100;
   1:  PR[GP1:91,1] = PR[GP1:90,1] + -55.176;
   1:  PR[GP1:91,2] = PR[GP1:90,2] + 31.207;
   1:L PR[91] 10mm/sec CNT100;
   1:  PR[GP1:91,1] = PR[GP1:90,1] + -58.608;
   1:  PR[GP1:91,2] = PR[GP1:90,2] + 28.987;
   1:L PR[91] 10mm/sec CNT100;
   1:  PR[GP1:91,1] = PR[GP1:90,1] + -63.325;
   1:  PR[GP1:91,2] = PR[GP1:90,2] + 25.553;
   1:L PR[91] 10mm/sec CNT100;
   1:  PR[GP1:91,1] = PR[GP1:90,1] + -66.321;
   1:  PR[GP1:91,2] = PR[GP1:90,2] + 22.495;
   1:L PR[91] 10mm/sec CNT100;
   1:  PR[GP1:91,1] = PR[GP1:90,1] + -68.600;
   1:  PR[GP1:91,2] = PR[GP1:90,2] + 18.808;
   1:L PR[91] 10mm/sec CNT100;
   1:  PR[GP1:91,1] = PR[GP1:90,1] + -71.564;
   1:  PR[GP1:91,2] = PR[GP1:90,2] + 14.125;
   1:L PR[91] 10mm/sec CNT100;
   1:  PR[GP1:91,1] = PR[GP1:90,1] + -72.998;
   1:  PR[GP1:91,2] = PR[GP1:90,2] + 9.969;
   1:L PR[91] 10mm/sec CNT100;
   1:  PR[GP1:91,1] = PR[GP1:90,1] + -73.494;
   1:  PR[GP1:91,2] = PR[GP1:90,2] + 5.507;
   1:L PR[91] 10mm/sec CNT100;
   1:  PR[GP1:91,1] = PR[GP1:90,1] + -74.488;
   1:  PR[GP1:91,2] = PR[GP1:90,2] + 0.256;
   1:L PR[91] 10mm/sec CNT100;
   1:  PR[GP1:91,1] = PR[GP1:90,1] + -73.986;
   1:  PR[GP1:91,2] = PR[GP1:90,2] + -4.260;
   1:L PR[91] 10mm/sec CNT100;
   1:  PR[GP1:91,1] = PR[GP1:90,1] + -73.005;
   1:  PR[GP1:91,2] = PR[GP1:90,2] + -9.388;
   1:L PR[91] 10mm/sec CNT100;
   1:  PR[GP1:91,1] = PR[GP1:90,1] + -71.563;
   1:  PR[GP1:91,2] = PR[GP1:90,2] + -13.570;
   1:L PR[91] 10mm/sec CNT100;
   1:  PR[GP1:91,1] = PR[GP1:90,1] + -69.216;
   1:  PR[GP1:91,2] = PR[GP1:90,2] + -17.367;
   1:L PR[91] 10mm/sec CNT100;
   1:  PR[GP1:91,1] = PR[GP1:90,1] + -66.323;
   1:  PR[GP1:91,2] = PR[GP1:90,2] + -21.934;
   1:L PR[91] 10mm/sec CNT100;
   1:  PR[GP1:91,1] = PR[GP1:90,1] + -63.336;
   1:  PR[GP1:91,2] = PR[GP1:90,2] + -24.983;
   1:L PR[91] 10mm/sec CNT100;
   1:  PR[GP1:91,1] = PR[GP1:90,1] + -59.685;
   1:  PR[GP1:91,2] = PR[GP1:90,2] + -27.345;
   1:L PR[91] 10mm/sec CNT100;
   1:  PR[GP1:91,1] = PR[GP1:90,1] + -55.160;
   1:  PR[GP1:91,2] = PR[GP1:90,2] + -30.655;
   1:L PR[91] 10mm/sec CNT100;
   1:  PR[GP1:91,1] = PR[GP1:90,1] + -51.354;
   1:  PR[GP1:91,2] = PR[GP1:90,2] + -32.056;
   1:L PR[91] 10mm/sec CNT100;
   1:  PR[GP1:91,1] = PR[GP1:90,1] + -45.324;
   1:  PR[GP1:91,2] = PR[GP1:90,2] + -33.620;
   1:L PR[91] 10mm/sec CNT100;
   1:  PR[GP1:91,1] = PR[GP1:90,1] + -41.609;
   1:  PR[GP1:91,2] = PR[GP1:90,2] + -34.111;
   1:L PR[91] 10mm/sec CNT100;
   1:  PR[GP1:91,1] = PR[GP1:90,1] + -37.849;
   1:  PR[GP1:91,2] = PR[GP1:90,2] + -33.771;
   1:L PR[91] 10mm/sec CNT100;
   1:  PR[GP1:91,1] = PR[GP1:90,1] + -31.185;
   1:  PR[GP1:91,2] = PR[GP1:90,2] + -32.967;
   1:L PR[91] 10mm/sec CNT100;
   1:  PR[GP1:91,1] = PR[GP1:90,1] + -28.013;
   1:  PR[GP1:91,2] = PR[GP1:90,2] + -31.945;
   1:L PR[91] 10mm/sec CNT100;
   1:  PR[GP1:91,1] = PR[GP1:90,1] + -25.082;
   1:  PR[GP1:91,2] = PR[GP1:90,2] + -30.216;
   1:L PR[91] 10mm/sec CNT100;
   1:  PR[GP1:91,1] = PR[GP1:90,1] + -18.681;
   1:  PR[GP1:91,2] = PR[GP1:90,2] + -26.782;
   1:L PR[91] 10mm/sec CNT100;
   1:  PR[GP1:91,1] = PR[GP1:90,1] + -16.553;
   1:  PR[GP1:91,2] = PR[GP1:90,2] + -24.782;
   1:L PR[91] 10mm/sec CNT100;
   1:  PR[GP1:91,1] = PR[GP1:90,1] + -11.249;
   1:  PR[GP1:91,2] = PR[GP1:90,2] + -18.495;
   1:L PR[91] 10mm/sec CNT100;
   1:  PR[GP1:91,1] = PR[GP1:90,1] + -9.810;
   1:  PR[GP1:91,2] = PR[GP1:90,2] + -16.368;
   1:L PR[91] 10mm/sec CNT100;
   1:  PR[GP1:91,1] = PR[GP1:90,1] + -8.867;
   1:  PR[GP1:91,2] = PR[GP1:90,2] + -13.961;
   1:L PR[91] 10mm/sec CNT100;
   1:  PR[GP1:91,1] = PR[GP1:90,1] + -6.098;
   1:  PR[GP1:91,2] = PR[GP1:90,2] + -5.804;
   1:L PR[91] 10mm/sec CNT100;
   1:  PR[GP1:91,1] = PR[GP1:90,1] + -5.752;
   1:  PR[GP1:91,2] = PR[GP1:90,2] + -3.548;
   1:L PR[91] 10mm/sec CNT100;
   1:  PR[GP1:91,1] = PR[GP1:90,1] + -5.962;
   1:  PR[GP1:91,2] = PR[GP1:90,2] + -2.808;
   1:L PR[91] 10mm/sec CNT100;
   1:  PR[GP1:91,1] = PR[GP1:90,1] + 5.165;
   1:L PR[91] 10mm/sec CNT100;
   1:  PR[GP1:91,1] = PR[GP1:90,1] + 5.451;
   1:  PR[GP1:91,2] = PR[GP1:90,2] + -5.436;
   1:  PR[GP1:91,3] = PR[GP1:90,3] + 13.725;
   1:L PR[91] 10mm/sec CNT100;
   1:  PR[GP1:91,1] = PR[GP1:90,1] + 6.087;
   1:  PR[GP1:91,2] = PR[GP1:90,2] + -7.060;
   1:L PR[91] 10mm/sec CNT100;
   1:  PR[GP1:91,1] = PR[GP1:90,1] + 9.288;
   1:  PR[GP1:91,2] = PR[GP1:90,2] + -16.454;
   1:L PR[91] 10mm/sec CNT100;
   1:  PR[GP1:91,1] = PR[GP1:90,1] + 10.359;
   1:  PR[GP1:91,2] = PR[GP1:90,2] + -18.037;
   1:L PR[91] 10mm/sec CNT100;
   1:  PR[GP1:91,1] = PR[GP1:90,1] + 16.340;
   1:  PR[GP1:91,2] = PR[GP1:90,2] + -25.133;
   1:L PR[91] 10mm/sec CNT100;
   1:  PR[GP1:91,1] = PR[GP1:90,1] + 18.042;
   1:  PR[GP1:91,2] = PR[GP1:90,2] + -26.733;
   1:L PR[91] 10mm/sec CNT100;
   1:  PR[GP1:91,1] = PR[GP1:90,1] + 20.074;
   1:  PR[GP1:91,2] = PR[GP1:90,2] + -27.931;
   1:L PR[91] 10mm/sec CNT100;
   1:  PR[GP1:91,1] = PR[GP1:90,1] + 27.706;
   1:  PR[GP1:91,2] = PR[GP1:90,2] + -32.048;
   1:L PR[91] 10mm/sec CNT100;
   1:  PR[GP1:91,1] = PR[GP1:90,1] + 30.364;
   1:  PR[GP1:91,2] = PR[GP1:90,2] + -32.904;
   1:L PR[91] 10mm/sec CNT100;
   1:  PR[GP1:91,1] = PR[GP1:90,1] + 33.209;
   1:  PR[GP1:91,2] = PR[GP1:90,2] + -33.161;
   1:L PR[91] 10mm/sec CNT100;
   1:  PR[GP1:91,1] = PR[GP1:90,1] + 41.169;
   1:  PR[GP1:91,2] = PR[GP1:90,2] + -34.110;
   1:L PR[91] 10mm/sec CNT100;
   1:  PR[GP1:91,1] = PR[GP1:90,1] + 44.387;
   1:  PR[GP1:91,2] = PR[GP1:90,2] + -33.685;
   1:L PR[91] 10mm/sec CNT100;
   1:  PR[GP1:91,1] = PR[GP1:90,1] + 51.191;
   1:  PR[GP1:91,2] = PR[GP1:90,2] + -31.921;
   1:L PR[91] 10mm/sec CNT100;
   1:  PR[GP1:91,1] = PR[GP1:90,1] + 54.590;
   1:  PR[GP1:91,2] = PR[GP1:90,2] + -30.670;
   1:L PR[91] 10mm/sec CNT100;
   1:  PR[GP1:91,1] = PR[GP1:90,1] + 57.641;
   1:  PR[GP1:91,2] = PR[GP1:90,2] + -28.695;
   1:L PR[91] 10mm/sec CNT100;
   1:  PR[GP1:91,1] = PR[GP1:90,1] + 62.964;
   1:  PR[GP1:91,2] = PR[GP1:90,2] + -24.821;
   1:L PR[91] 10mm/sec CNT100;
   1:  PR[GP1:91,1] = PR[GP1:90,1] + 65.664;
   1:  PR[GP1:91,2] = PR[GP1:90,2] + -22.065;
   1:L PR[91] 10mm/sec CNT100;
   1:  PR[GP1:91,1] = PR[GP1:90,1] + 67.720;
   1:  PR[GP1:91,2] = PR[GP1:90,2] + -18.738;
   1:L PR[91] 10mm/sec CNT100;
   1:  PR[GP1:91,1] = PR[GP1:90,1] + 71.066;
   1:  PR[GP1:91,2] = PR[GP1:90,2] + -13.455;
   1:L PR[91] 10mm/sec CNT100;
   1:  PR[GP1:91,1] = PR[GP1:90,1] + 72.367;
   1:  PR[GP1:91,2] = PR[GP1:90,2] + -9.683;
   1:L PR[91] 10mm/sec CNT100;
   1:  PR[GP1:91,1] = PR[GP1:90,1] + 72.818;
   1:  PR[GP1:91,2] = PR[GP1:90,2] + -5.625;
   1:L PR[91] 10mm/sec CNT100;
   1:  PR[GP1:91,1] = PR[GP1:90,1] + 73.941;
   1:  PR[GP1:91,2] = PR[GP1:90,2] + 0.302;
   1:L PR[91] 10mm/sec CNT100;
   1:  PR[GP1:91,1] = PR[GP1:90,1] + 73.482;
   1:  PR[GP1:91,2] = PR[GP1:90,2] + 4.430;
   1:L PR[91] 10mm/sec CNT100;
   1:  PR[GP1:91,1] = PR[GP1:90,1] + 72.375;
   1:  PR[GP1:91,2] = PR[GP1:90,2] + 10.219;
   1:L PR[91] 10mm/sec CNT100;
   1:  PR[GP1:91,1] = PR[GP1:90,1] + 71.065;
   1:  PR[GP1:91,2] = PR[GP1:90,2] + 14.017;
   1:L PR[91] 10mm/sec CNT100;
   1:  PR[GP1:91,1] = PR[GP1:90,1] + 68.931;
   1:  PR[GP1:91,2] = PR[GP1:90,2] + 17.468;
   1:L PR[91] 10mm/sec CNT100;
   1:  PR[GP1:91,1] = PR[GP1:90,1] + 65.666;
   1:  PR[GP1:91,2] = PR[GP1:90,2] + 22.621;
   1:L PR[91] 10mm/sec CNT100;
   1:  PR[GP1:91,1] = PR[GP1:90,1] + 62.976;
   1:  PR[GP1:91,2] = PR[GP1:90,2] + 25.367;
   1:L PR[91] 10mm/sec CNT100;
   1:  PR[GP1:91,1] = PR[GP1:90,1] + 59.680;
   1:  PR[GP1:91,2] = PR[GP1:90,2] + 27.499;
   1:L PR[91] 10mm/sec CNT100;
   1:  PR[GP1:91,1] = PR[GP1:90,1] + 54.573;
   1:  PR[GP1:91,2] = PR[GP1:90,2] + 31.234;
   1:L PR[91] 10mm/sec CNT100;
   1:  PR[GP1:91,1] = PR[GP1:90,1] + 51.191;
   1:  PR[GP1:91,2] = PR[GP1:90,2] + 32.479;
   1:L PR[91] 10mm/sec CNT100;
   1:  PR[GP1:91,1] = PR[GP1:90,1] + 44.387;
   1:  PR[GP1:91,2] = PR[GP1:90,2] + 34.243;
   1:L PR[91] 10mm/sec CNT100;
   1:  PR[GP1:91,1] = PR[GP1:90,1] + 41.161;
   1:  PR[GP1:91,2] = PR[GP1:90,2] + 34.669;
   1:L PR[91] 10mm/sec CNT100;
   1:  PR[GP1:91,1] = PR[GP1:90,1] + 37.891;
   1:  PR[GP1:91,2] = PR[GP1:90,2] + 34.374;
   1:L PR[91] 10mm/sec CNT100;
   1:  PR[GP1:91,1] = PR[GP1:90,1] + 30.373;
   1:  PR[GP1:91,2] = PR[GP1:90,2] + 33.465;
   1:L PR[91] 10mm/sec CNT100;
   1:  PR[GP1:91,1] = PR[GP1:90,1] + 27.718;
   1:  PR[GP1:91,2] = PR[GP1:90,2] + 32.610;
   1:L PR[91] 10mm/sec CNT100;
   1:  PR[GP1:91,1] = PR[GP1:90,1] + 25.255;
   1:  PR[GP1:91,2] = PR[GP1:90,2] + 31.157;
   1:L PR[91] 10mm/sec CNT100;
   1:  PR[GP1:91,1] = PR[GP1:90,1] + 18.033;
   1:  PR[GP1:91,2] = PR[GP1:90,2] + 27.282;
   1:L PR[91] 10mm/sec CNT100;
   1:  PR[GP1:91,1] = PR[GP1:90,1] + 16.340;
   1:  PR[GP1:91,2] = PR[GP1:90,2] + 25.691;
   1:L PR[91] 10mm/sec CNT100;
   1:  PR[GP1:91,1] = PR[GP1:90,1] + 10.359;
   1:  PR[GP1:91,2] = PR[GP1:90,2] + 18.595;
   1:L PR[91] 10mm/sec CNT100;
   1:  PR[GP1:91,1] = PR[GP1:90,1] + 9.280;
   1:  PR[GP1:91,2] = PR[GP1:90,2] + 17.001;
   1:L PR[91] 10mm/sec CNT100;
   1:  PR[GP1:91,1] = PR[GP1:90,1] + 8.572;
   1:  PR[GP1:91,2] = PR[GP1:90,2] + 15.192;
   1:L PR[91] 10mm/sec CNT100;
   1:  PR[GP1:91,1] = PR[GP1:90,1] + 5.450;
   1:  PR[GP1:91,2] = PR[GP1:90,2] + 6.000;
   1:L PR[91] 10mm/sec CNT100;
   1:  PR[GP1:91,1] = PR[GP1:90,1] + 5.206;
   1:  PR[GP1:91,2] = PR[GP1:90,2] + 4.404;
   1:L PR[91] 10mm/sec CNT100;
   1:  PR[GP1:91,1] = PR[GP1:90,1] + 5.409;
   1:  PR[GP1:91,2] = PR[GP1:90,2] + 3.691;
   1:L PR[91] 10mm/sec CNT100;
   1:  PR[GP1:91,1] = PR[GP1:90,1] + -5.665;
   1:L PR[91] 10mm/sec CNT100;
   1:  PR[GP1:91,1] = PR[GP1:90,1] + -5.977;
   1:  PR[GP1:91,2] = PR[GP1:90,2] + 5.994;
   1:L PR[91] 10mm/sec CNT100;
   1:  PR[GP1:91,1] = PR[GP1:90,1] + -6.613;
   1:  PR[GP1:91,2] = PR[GP1:90,2] + 7.617;
   1:L PR[91] 10mm/sec CNT100;
   1:  PR[GP1:91,1] = PR[GP1:90,1] + -9.817;
   1:  PR[GP1:91,2] = PR[GP1:90,2] + 17.019;
   1:L PR[91] 10mm/sec CNT100;
   1:  PR[GP1:91,1] = PR[GP1:90,1] + -10.888;
   1:  PR[GP1:91,2] = PR[GP1:90,2] + 18.602;
   1:L PR[91] 10mm/sec CNT100;
   1:  PR[GP1:91,1] = PR[GP1:90,1] + -16.870;
   1:  PR[GP1:91,2] = PR[GP1:90,2] + 25.693;
   1:L PR[91] 10mm/sec CNT100;
   1:  PR[GP1:91,1] = PR[GP1:90,1] + -18.572;
   1:  PR[GP1:91,2] = PR[GP1:90,2] + 27.293;
   1:L PR[91] 10mm/sec CNT100;
   1:  PR[GP1:91,1] = PR[GP1:90,1] + -20.604;
   1:  PR[GP1:91,2] = PR[GP1:90,2] + 28.492;
   1:L PR[91] 10mm/sec CNT100;
   1:  PR[GP1:91,1] = PR[GP1:90,1] + -28.236;
   1:  PR[GP1:91,2] = PR[GP1:90,2] + 32.608;
   1:L PR[91] 10mm/sec CNT100;
   1:  PR[GP1:91,1] = PR[GP1:90,1] + -30.894;
   1:  PR[GP1:91,2] = PR[GP1:90,2] + 33.464;
   1:L PR[91] 10mm/sec CNT100;
   1:  PR[GP1:91,1] = PR[GP1:90,1] + -33.739;
   1:  PR[GP1:91,2] = PR[GP1:90,2] + 33.721;
   1:L PR[91] 10mm/sec CNT100;
   1:  PR[GP1:91,1] = PR[GP1:90,1] + -41.698;
   1:  PR[GP1:91,2] = PR[GP1:90,2] + 34.668;
   1:L PR[91] 10mm/sec CNT100;
   1:  PR[GP1:91,1] = PR[GP1:90,1] + -44.916;
   1:  PR[GP1:91,2] = PR[GP1:90,2] + 34.243;
   1:L PR[91] 10mm/sec CNT100;
   1:  PR[GP1:91,1] = PR[GP1:90,1] + -51.719;
   1:  PR[GP1:91,2] = PR[GP1:90,2] + 32.478;
   1:L PR[91] 10mm/sec CNT100;
   1:  PR[GP1:91,1] = PR[GP1:90,1] + -55.117;
   1:  PR[GP1:91,2] = PR[GP1:90,2] + 31.227;
   1:L PR[91] 10mm/sec CNT100;
   1:  PR[GP1:91,1] = PR[GP1:90,1] + -58.169;
   1:  PR[GP1:91,2] = PR[GP1:90,2] + 29.253;
   1:L PR[91] 10mm/sec CNT100;
   1:  PR[GP1:91,1] = PR[GP1:90,1] + -63.491;
   1:  PR[GP1:91,2] = PR[GP1:90,2] + 25.378;
   1:L PR[91] 10mm/sec CNT100;
   1:  PR[GP1:91,1] = PR[GP1:90,1] + -66.191;
   1:  PR[GP1:91,2] = PR[GP1:90,2] + 22.622;
   1:L PR[91] 10mm/sec CNT100;
   1:  PR[GP1:91,1] = PR[GP1:90,1] + -68.247;
   1:  PR[GP1:91,2] = PR[GP1:90,2] + 19.295;
   1:L PR[91] 10mm/sec CNT100;
   1:  PR[GP1:91,1] = PR[GP1:90,1] + -71.592;
   1:  PR[GP1:91,2] = PR[GP1:90,2] + 14.012;
   1:L PR[91] 10mm/sec CNT100;
   1:  PR[GP1:91,1] = PR[GP1:90,1] + -72.893;
   1:  PR[GP1:91,2] = PR[GP1:90,2] + 10.239;
   1:L PR[91] 10mm/sec CNT100;
   1:  PR[GP1:91,1] = PR[GP1:90,1] + -73.345;
   1:  PR[GP1:91,2] = PR[GP1:90,2] + 6.181;
   1:L PR[91] 10mm/sec CNT100;
   1:  PR[GP1:91,1] = PR[GP1:90,1] + -74.467;
   1:  PR[GP1:91,2] = PR[GP1:90,2] + 0.256;
   1:L PR[91] 10mm/sec CNT100;
   1:  PR[GP1:91,1] = PR[GP1:90,1] + -74.008;
   1:  PR[GP1:91,2] = PR[GP1:90,2] + -3.872;
   1:L PR[91] 10mm/sec CNT100;
   1:  PR[GP1:91,1] = PR[GP1:90,1] + -72.901;
   1:  PR[GP1:91,2] = PR[GP1:90,2] + -9.659;
   1:L PR[91] 10mm/sec CNT100;
   1:  PR[GP1:91,1] = PR[GP1:90,1] + -71.591;
   1:  PR[GP1:91,2] = PR[GP1:90,2] + -13.457;
   1:L PR[91] 10mm/sec CNT100;
   1:  PR[GP1:91,1] = PR[GP1:90,1] + -69.458;
   1:  PR[GP1:91,2] = PR[GP1:90,2] + -16.908;
   1:L PR[91] 10mm/sec CNT100;
   1:  PR[GP1:91,1] = PR[GP1:90,1] + -66.193;
   1:  PR[GP1:91,2] = PR[GP1:90,2] + -22.062;
   1:L PR[91] 10mm/sec CNT100;
   1:  PR[GP1:91,1] = PR[GP1:90,1] + -63.503;
   1:  PR[GP1:91,2] = PR[GP1:90,2] + -24.809;
   1:L PR[91] 10mm/sec CNT100;
   1:  PR[GP1:91,1] = PR[GP1:90,1] + -60.207;
   1:  PR[GP1:91,2] = PR[GP1:90,2] + -26.941;
   1:L PR[91] 10mm/sec CNT100;
   1:  PR[GP1:91,1] = PR[GP1:90,1] + -55.101;
   1:  PR[GP1:91,2] = PR[GP1:90,2] + -30.675;
   1:L PR[91] 10mm/sec CNT100;
   1:  PR[GP1:91,1] = PR[GP1:90,1] + -51.719;
   1:  PR[GP1:91,2] = PR[GP1:90,2] + -31.920;
   1:L PR[91] 10mm/sec CNT100;
   1:  PR[GP1:91,1] = PR[GP1:90,1] + -44.916;
   1:  PR[GP1:91,2] = PR[GP1:90,2] + -33.685;
   1:L PR[91] 10mm/sec CNT100;
   1:  PR[GP1:91,1] = PR[GP1:90,1] + -41.690;
   1:  PR[GP1:91,2] = PR[GP1:90,2] + -34.111;
   1:L PR[91] 10mm/sec CNT100;
   1:  PR[GP1:91,1] = PR[GP1:90,1] + -38.420;
   1:  PR[GP1:91,2] = PR[GP1:90,2] + -33.816;
   1:L PR[91] 10mm/sec CNT100;
   1:  PR[GP1:91,1] = PR[GP1:90,1] + -30.903;
   1:  PR[GP1:91,2] = PR[GP1:90,2] + -32.908;
   1:L PR[91] 10mm/sec CNT100;
   1:  PR[GP1:91,1] = PR[GP1:90,1] + -28.247;
   1:  PR[GP1:91,2] = PR[GP1:90,2] + -32.053;
   1:L PR[91] 10mm/sec CNT100;
   1:  PR[GP1:91,1] = PR[GP1:90,1] + -25.784;
   1:  PR[GP1:91,2] = PR[GP1:90,2] + -30.600;
   1:L PR[91] 10mm/sec CNT100;
   1:  PR[GP1:91,1] = PR[GP1:90,1] + -18.563;
   1:  PR[GP1:91,2] = PR[GP1:90,2] + -26.726;
   1:L PR[91] 10mm/sec CNT100;
   1:  PR[GP1:91,1] = PR[GP1:90,1] + -16.870;
   1:  PR[GP1:91,2] = PR[GP1:90,2] + -25.134;
   1:L PR[91] 10mm/sec CNT100;
   1:  PR[GP1:91,1] = PR[GP1:90,1] + -10.888;
   1:  PR[GP1:91,2] = PR[GP1:90,2] + -18.044;
   1:L PR[91] 10mm/sec CNT100;
   1:  PR[GP1:91,1] = PR[GP1:90,1] + -9.809;
   1:  PR[GP1:91,2] = PR[GP1:90,2] + -16.449;
   1:L PR[91] 10mm/sec CNT100;
   1:  PR[GP1:91,1] = PR[GP1:90,1] + -9.101;
   1:  PR[GP1:91,2] = PR[GP1:90,2] + -14.640;
   1:L PR[91] 10mm/sec CNT100;
   1:  PR[GP1:91,1] = PR[GP1:90,1] + -5.977;
   1:  PR[GP1:91,2] = PR[GP1:90,2] + -5.442;
   1:L PR[91] 10mm/sec CNT100;
   1:  PR[GP1:91,1] = PR[GP1:90,1] + -5.733;
   1:  PR[GP1:91,2] = PR[GP1:90,2] + -3.845;
   1:L PR[91] 10mm/sec CNT100;
   1:  PR[GP1:91,1] = PR[GP1:90,1] + -5.935;
   1:  PR[GP1:91,2] = PR[GP1:90,2] + -3.133;
   1:L PR[91] 10mm/sec CNT100;
   1:  PR[GP1:91,1] = PR[GP1:90,1] + 5.138;
   1:L PR[91] 10mm/sec CNT100;
   1:  PR[GP1:91,1] = PR[GP1:90,1] + 5.330;
   1:  PR[GP1:91,2] = PR[GP1:90,2] + -5.074;
   1:  PR[GP1:91,3] = PR[GP1:90,3] + 14.335;
   1:L PR[91] 10mm/sec CNT100;
   1:  PR[GP1:91,1] = PR[GP1:90,1] + 5.722;
   1:  PR[GP1:91,2] = PR[GP1:90,2] + -6.076;
   1:L PR[91] 10mm/sec CNT100;
   1:  PR[GP1:91,1] = PR[GP1:90,1] + 9.287;
   1:  PR[GP1:91,2] = PR[GP1:90,2] + -16.534;
   1:L PR[91] 10mm/sec CNT100;
   1:  PR[GP1:91,1] = PR[GP1:90,1] + 9.997;
   1:  PR[GP1:91,2] = PR[GP1:90,2] + -17.585;
   1:L PR[91] 10mm/sec CNT100;
   1:  PR[GP1:91,1] = PR[GP1:90,1] + 16.657;
   1:  PR[GP1:91,2] = PR[GP1:90,2] + -25.485;
   1:L PR[91] 10mm/sec CNT100;
   1:  PR[GP1:91,1] = PR[GP1:90,1] + 17.924;
   1:  PR[GP1:91,2] = PR[GP1:90,2] + -26.676;
   1:L PR[91] 10mm/sec CNT100;
   1:  PR[GP1:91,1] = PR[GP1:90,1] + 19.442;
   1:  PR[GP1:91,2] = PR[GP1:90,2] + -27.572;
   1:L PR[91] 10mm/sec CNT100;
   1:  PR[GP1:91,1] = PR[GP1:90,1] + 27.940;
   1:  PR[GP1:91,2] = PR[GP1:90,2] + -32.156;
   1:L PR[91] 10mm/sec CNT100;
   1:  PR[GP1:91,1] = PR[GP1:90,1] + 30.082;
   1:  PR[GP1:91,2] = PR[GP1:90,2] + -32.845;
   1:L PR[91] 10mm/sec CNT100;
   1:  PR[GP1:91,1] = PR[GP1:90,1] + 32.386;
   1:  PR[GP1:91,2] = PR[GP1:90,2] + -33.054;
   1:L PR[91] 10mm/sec CNT100;
   1:  PR[GP1:91,1] = PR[GP1:90,1] + 41.250;
   1:  PR[GP1:91,2] = PR[GP1:90,2] + -34.110;
   1:L PR[91] 10mm/sec CNT100;
   1:  PR[GP1:91,1] = PR[GP1:90,1] + 43.980;
   1:  PR[GP1:91,2] = PR[GP1:90,2] + -33.750;
   1:L PR[91] 10mm/sec CNT100;
   1:  PR[GP1:91,1] = PR[GP1:90,1] + 51.556;
   1:  PR[GP1:91,2] = PR[GP1:90,2] + -31.785;
   1:L PR[91] 10mm/sec CNT100;
   1:  PR[GP1:91,1] = PR[GP1:90,1] + 54.530;
   1:  PR[GP1:91,2] = PR[GP1:90,2] + -30.690;
   1:L PR[91] 10mm/sec CNT100;
   1:  PR[GP1:91,1] = PR[GP1:90,1] + 57.202;
   1:  PR[GP1:91,2] = PR[GP1:90,2] + -28.961;
   1:L PR[91] 10mm/sec CNT100;
   1:  PR[GP1:91,1] = PR[GP1:90,1] + 63.130;
   1:  PR[GP1:91,2] = PR[GP1:90,2] + -24.646;
   1:L PR[91] 10mm/sec CNT100;
   1:  PR[GP1:91,1] = PR[GP1:90,1] + 65.534;
   1:  PR[GP1:91,2] = PR[GP1:90,2] + -22.193;
   1:L PR[91] 10mm/sec CNT100;
   1:  PR[GP1:91,1] = PR[GP1:90,1] + 67.368;
   1:  PR[GP1:91,2] = PR[GP1:90,2] + -19.226;
   1:L PR[91] 10mm/sec CNT100;
   1:  PR[GP1:91,1] = PR[GP1:90,1] + 71.094;
   1:  PR[GP1:91,2] = PR[GP1:90,2] + -13.342;
   1:L PR[91] 10mm/sec CNT100;
   1:  PR[GP1:91,1] = PR[GP1:90,1] + 72.263;
   1:  PR[GP1:91,2] = PR[GP1:90,2] + -9.954;
   1:L PR[91] 10mm/sec CNT100;
   1:  PR[GP1:91,1] = PR[GP1:90,1] + 72.669;
   1:  PR[GP1:91,2] = PR[GP1:90,2] + -6.299;
   1:L PR[91] 10mm/sec CNT100;
   1:  PR[GP1:91,1] = PR[GP1:90,1] + 73.919;
   1:  PR[GP1:91,2] = PR[GP1:90,2] + 0.302;
   1:L PR[91] 10mm/sec CNT100;
   1:  PR[GP1:91,1] = PR[GP1:90,1] + 73.504;
   1:  PR[GP1:91,2] = PR[GP1:90,2] + 4.042;
   1:L PR[91] 10mm/sec CNT100;
   1:  PR[GP1:91,1] = PR[GP1:90,1] + 72.270;
   1:  PR[GP1:91,2] = PR[GP1:90,2] + 10.490;
   1:L PR[91] 10mm/sec CNT100;
   1:  PR[GP1:91,1] = PR[GP1:90,1] + 71.093;
   1:  PR[GP1:91,2] = PR[GP1:90,2] + 13.904;
   1:L PR[91] 10mm/sec CNT100;
   1:  PR[GP1:91,1] = PR[GP1:90,1] + 69.173;
   1:  PR[GP1:91,2] = PR[GP1:90,2] + 17.009;
   1:L PR[91] 10mm/sec CNT100;
   1:  PR[GP1:91,1] = PR[GP1:90,1] + 65.536;
   1:  PR[GP1:91,2] = PR[GP1:90,2] + 22.748;
   1:L PR[91] 10mm/sec CNT100;
   1:  PR[GP1:91,1] = PR[GP1:90,1] + 63.142;
   1:  PR[GP1:91,2] = PR[GP1:90,2] + 25.193;
   1:L PR[91] 10mm/sec CNT100;
   1:  PR[GP1:91,1] = PR[GP1:90,1] + 60.202;
   1:  PR[GP1:91,2] = PR[GP1:90,2] + 27.095;
   1:L PR[91] 10mm/sec CNT100;
   1:  PR[GP1:91,1] = PR[GP1:90,1] + 54.514;
   1:  PR[GP1:91,2] = PR[GP1:90,2] + 31.254;
   1:L PR[91] 10mm/sec CNT100;
   1:  PR[GP1:91,1] = PR[GP1:90,1] + 51.556;
   1:  PR[GP1:91,2] = PR[GP1:90,2] + 32.343;
   1:L PR[91] 10mm/sec CNT100;
   1:  PR[GP1:91,1] = PR[GP1:90,1] + 43.980;
   1:  PR[GP1:91,2] = PR[GP1:90,2] + 34.308;
   1:L PR[91] 10mm/sec CNT100;
   1:  PR[GP1:91,1] = PR[GP1:90,1] + 41.241;
   1:  PR[GP1:91,2] = PR[GP1:90,2] + 34.669;
   1:L PR[91] 10mm/sec CNT100;
   1:  PR[GP1:91,1] = PR[GP1:90,1] + 38.463;
   1:  PR[GP1:91,2] = PR[GP1:90,2] + 34.418;
   1:L PR[91] 10mm/sec CNT100;
   1:  PR[GP1:91,1] = PR[GP1:90,1] + 30.091;
   1:  PR[GP1:91,2] = PR[GP1:90,2] + 33.406;
   1:L PR[91] 10mm/sec CNT100;
   1:  PR[GP1:91,1] = PR[GP1:90,1] + 27.951;
   1:  PR[GP1:91,2] = PR[GP1:90,2] + 32.717;
   1:L PR[91] 10mm/sec CNT100;
   1:  PR[GP1:91,1] = PR[GP1:90,1] + 25.956;
   1:  PR[GP1:91,2] = PR[GP1:90,2] + 31.540;
   1:L PR[91] 10mm/sec CNT100;
   1:  PR[GP1:91,1] = PR[GP1:90,1] + 17.915;
   1:  PR[GP1:91,2] = PR[GP1:90,2] + 27.226;
   1:L PR[91] 10mm/sec CNT100;
   1:  PR[GP1:91,1] = PR[GP1:90,1] + 16.657;
   1:  PR[GP1:91,2] = PR[GP1:90,2] + 26.043;
   1:L PR[91] 10mm/sec CNT100;
   1:  PR[GP1:91,1] = PR[GP1:90,1] + 9.997;
   1:  PR[GP1:91,2] = PR[GP1:90,2] + 18.143;
   1:L PR[91] 10mm/sec CNT100;
   1:  PR[GP1:91,1] = PR[GP1:90,1] + 9.279;
   1:  PR[GP1:91,2] = PR[GP1:90,2] + 17.081;
   1:L PR[91] 10mm/sec CNT100;
   1:  PR[GP1:91,1] = PR[GP1:90,1] + 8.805;
   1:  PR[GP1:91,2] = PR[GP1:90,2] + 15.871;
   1:L PR[91] 10mm/sec CNT100;
   1:  PR[GP1:91,1] = PR[GP1:90,1] + 5.330;
   1:  PR[GP1:91,2] = PR[GP1:90,2] + 5.637;
   1:L PR[91] 10mm/sec CNT100;
   1:  PR[GP1:91,1] = PR[GP1:90,1] + 5.186;
   1:  PR[GP1:91,2] = PR[GP1:90,2] + 4.701;
   1:L PR[91] 10mm/sec CNT100;
   1:  PR[GP1:91,1] = PR[GP1:90,1] + 5.381;
   1:  PR[GP1:91,2] = PR[GP1:90,2] + 4.016;
   1:L PR[91] 10mm/sec CNT100;
   1:  PR[GP1:91,1] = PR[GP1:90,1] + -5.637;
   1:L PR[91] 10mm/sec CNT100;
   1:  PR[GP1:91,1] = PR[GP1:90,1] + -5.857;
   1:  PR[GP1:91,2] = PR[GP1:90,2] + 5.632;
   1:L PR[91] 10mm/sec CNT100;
   1:  PR[GP1:91,1] = PR[GP1:90,1] + -6.249;
   1:  PR[GP1:91,2] = PR[GP1:90,2] + 6.633;
   1:L PR[91] 10mm/sec CNT100;
   1:  PR[GP1:91,1] = PR[GP1:90,1] + -9.816;
   1:  PR[GP1:91,2] = PR[GP1:90,2] + 17.100;
   1:L PR[91] 10mm/sec CNT100;
   1:  PR[GP1:91,1] = PR[GP1:90,1] + -10.527;
   1:  PR[GP1:91,2] = PR[GP1:90,2] + 18.150;
   1:L PR[91] 10mm/sec CNT100;
   1:  PR[GP1:91,1] = PR[GP1:90,1] + -17.186;
   1:  PR[GP1:91,2] = PR[GP1:90,2] + 26.045;
   1:L PR[91] 10mm/sec CNT100;
   1:  PR[GP1:91,1] = PR[GP1:90,1] + -18.454;
   1:  PR[GP1:91,2] = PR[GP1:90,2] + 27.237;
   1:L PR[91] 10mm/sec CNT100;
   1:  PR[GP1:91,1] = PR[GP1:90,1] + -19.973;
   1:  PR[GP1:91,2] = PR[GP1:90,2] + 28.133;
   1:L PR[91] 10mm/sec CNT100;
   1:  PR[GP1:91,1] = PR[GP1:90,1] + -28.470;
   1:  PR[GP1:91,2] = PR[GP1:90,2] + 32.715;
   1:L PR[91] 10mm/sec CNT100;
   1:  PR[GP1:91,1] = PR[GP1:90,1] + -30.612;
   1:  PR[GP1:91,2] = PR[GP1:90,2] + 33.405;
   1:L PR[91] 10mm/sec CNT100;
   1:  PR[GP1:91,1] = PR[GP1:90,1] + -32.916;
   1:  PR[GP1:91,2] = PR[GP1:90,2] + 33.613;
   1:L PR[91] 10mm/sec CNT100;
   1:  PR[GP1:91,1] = PR[GP1:90,1] + -41.779;
   1:  PR[GP1:91,2] = PR[GP1:90,2] + 34.668;
   1:L PR[91] 10mm/sec CNT100;
   1:  PR[GP1:91,1] = PR[GP1:90,1] + -44.509;
   1:  PR[GP1:91,2] = PR[GP1:90,2] + 34.307;
   1:L PR[91] 10mm/sec CNT100;
   1:  PR[GP1:91,1] = PR[GP1:90,1] + -52.084;
   1:  PR[GP1:91,2] = PR[GP1:90,2] + 32.342;
   1:L PR[91] 10mm/sec CNT100;
   1:  PR[GP1:91,1] = PR[GP1:90,1] + -55.059;
   1:  PR[GP1:91,2] = PR[GP1:90,2] + 31.247;
   1:L PR[91] 10mm/sec CNT100;
   1:  PR[GP1:91,1] = PR[GP1:90,1] + -57.731;
   1:  PR[GP1:91,2] = PR[GP1:90,2] + 29.519;
   1:L PR[91] 10mm/sec CNT100;
   1:  PR[GP1:91,1] = PR[GP1:90,1] + -63.657;
   1:  PR[GP1:91,2] = PR[GP1:90,2] + 25.204;
   1:L PR[91] 10mm/sec CNT100;
   1:  PR[GP1:91,1] = PR[GP1:90,1] + -66.061;
   1:  PR[GP1:91,2] = PR[GP1:90,2] + 22.750;
   1:L PR[91] 10mm/sec CNT100;
   1:  PR[GP1:91,1] = PR[GP1:90,1] + -67.895;
   1:  PR[GP1:91,2] = PR[GP1:90,2] + 19.783;
   1:L PR[91] 10mm/sec CNT100;
   1:  PR[GP1:91,1] = PR[GP1:90,1] + -71.620;
   1:  PR[GP1:91,2] = PR[GP1:90,2] + 13.899;
   1:L PR[91] 10mm/sec CNT100;
   1:  PR[GP1:91,1] = PR[GP1:90,1] + -72.789;
   1:  PR[GP1:91,2] = PR[GP1:90,2] + 10.510;
   1:L PR[91] 10mm/sec CNT100;
   1:  PR[GP1:91,1] = PR[GP1:90,1] + -73.196;
   1:  PR[GP1:91,2] = PR[GP1:90,2] + 6.855;
   1:L PR[91] 10mm/sec CNT100;
   1:  PR[GP1:91,1] = PR[GP1:90,1] + -74.446;
   1:  PR[GP1:91,2] = PR[GP1:90,2] + 0.256;
   1:L PR[91] 10mm/sec CNT100;
   1:  PR[GP1:91,1] = PR[GP1:90,1] + -74.030;
   1:  PR[GP1:91,2] = PR[GP1:90,2] + -3.484;
   1:L PR[91] 10mm/sec CNT100;
   1:  PR[GP1:91,1] = PR[GP1:90,1] + -72.797;
   1:  PR[GP1:91,2] = PR[GP1:90,2] + -9.930;
   1:L PR[91] 10mm/sec CNT100;
   1:  PR[GP1:91,1] = PR[GP1:90,1] + -71.619;
   1:  PR[GP1:91,2] = PR[GP1:90,2] + -13.344;
   1:L PR[91] 10mm/sec CNT100;
   1:  PR[GP1:91,1] = PR[GP1:90,1] + -69.700;
   1:  PR[GP1:91,2] = PR[GP1:90,2] + -16.449;
   1:L PR[91] 10mm/sec CNT100;
   1:  PR[GP1:91,1] = PR[GP1:90,1] + -66.063;
   1:  PR[GP1:91,2] = PR[GP1:90,2] + -22.190;
   1:L PR[91] 10mm/sec CNT100;
   1:  PR[GP1:91,1] = PR[GP1:90,1] + -63.669;
   1:  PR[GP1:91,2] = PR[GP1:90,2] + -24.634;
   1:L PR[91] 10mm/sec CNT100;
   1:  PR[GP1:91,1] = PR[GP1:90,1] + -60.729;
   1:  PR[GP1:91,2] = PR[GP1:90,2] + -26.536;
   1:L PR[91] 10mm/sec CNT100;
   1:  PR[GP1:91,1] = PR[GP1:90,1] + -55.042;
   1:  PR[GP1:91,2] = PR[GP1:90,2] + -30.695;
   1:L PR[91] 10mm/sec CNT100;
   1:  PR[GP1:91,1] = PR[GP1:90,1] + -52.084;
   1:  PR[GP1:91,2] = PR[GP1:90,2] + -31.784;
   1:L PR[91] 10mm/sec CNT100;
   1:  PR[GP1:91,1] = PR[GP1:90,1] + -44.509;
   1:  PR[GP1:91,2] = PR[GP1:90,2] + -33.749;
   1:L PR[91] 10mm/sec CNT100;
   1:  PR[GP1:91,1] = PR[GP1:90,1] + -41.770;
   1:  PR[GP1:91,2] = PR[GP1:90,2] + -34.111;
   1:L PR[91] 10mm/sec CNT100;
   1:  PR[GP1:91,1] = PR[GP1:90,1] + -38.992;
   1:  PR[GP1:91,2] = PR[GP1:90,2] + -33.860;
   1:L PR[91] 10mm/sec CNT100;
   1:  PR[GP1:91,1] = PR[GP1:90,1] + -30.620;
   1:  PR[GP1:91,2] = PR[GP1:90,2] + -32.850;
   1:L PR[91] 10mm/sec CNT100;
   1:  PR[GP1:91,1] = PR[GP1:90,1] + -28.481;
   1:  PR[GP1:91,2] = PR[GP1:90,2] + -32.161;
   1:L PR[91] 10mm/sec CNT100;
   1:  PR[GP1:91,1] = PR[GP1:90,1] + -26.485;
   1:  PR[GP1:91,2] = PR[GP1:90,2] + -30.983;
   1:L PR[91] 10mm/sec CNT100;
   1:  PR[GP1:91,1] = PR[GP1:90,1] + -18.445;
   1:  PR[GP1:91,2] = PR[GP1:90,2] + -26.670;
   1:L PR[91] 10mm/sec CNT100;
   1:  PR[GP1:91,1] = PR[GP1:90,1] + -17.186;
   1:  PR[GP1:91,2] = PR[GP1:90,2] + -25.487;
   1:L PR[91] 10mm/sec CNT100;
   1:  PR[GP1:91,1] = PR[GP1:90,1] + -10.527;
   1:  PR[GP1:91,2] = PR[GP1:90,2] + -17.592;
   1:L PR[91] 10mm/sec CNT100;
   1:  PR[GP1:91,1] = PR[GP1:90,1] + -9.808;
   1:  PR[GP1:91,2] = PR[GP1:90,2] + -16.530;
   1:L PR[91] 10mm/sec CNT100;
   1:  PR[GP1:91,1] = PR[GP1:90,1] + -9.334;
   1:  PR[GP1:91,2] = PR[GP1:90,2] + -15.320;
   1:L PR[91] 10mm/sec CNT100;
   1:  PR[GP1:91,1] = PR[GP1:90,1] + -5.856;
   1:  PR[GP1:91,2] = PR[GP1:90,2] + -5.079;
   1:L PR[91] 10mm/sec CNT100;
   1:  PR[GP1:91,1] = PR[GP1:90,1] + -5.713;
   1:  PR[GP1:91,2] = PR[GP1:90,2] + -4.143;
   1:L PR[91] 10mm/sec CNT100;
   1:  PR[GP1:91,1] = PR[GP1:90,1] + -5.908;
   1:  PR[GP1:91,2] = PR[GP1:90,2] + -3.458;
   1:L PR[91] 10mm/sec CNT100;
   1:  PR[GP1:91,1] = PR[GP1:90,1] + 5.111;
   1:L PR[91] 10mm/sec CNT100;
   1:  PR[GP1:91,1] = PR[GP1:90,1] + 5.209;
   1:  PR[GP1:91,2] = PR[GP1:90,2] + -4.712;
   1:  PR[GP1:91,3] = PR[GP1:90,3] + 14.945;
   1:L PR[91] 10mm/sec CNT100;
   1:  PR[GP1:91,1] = PR[GP1:90,1] + 5.358;
   1:  PR[GP1:91,2] = PR[GP1:90,2] + -5.092;
   1:L PR[91] 10mm/sec CNT100;
   1:  PR[GP1:91,1] = PR[GP1:90,1] + 9.285;
   1:  PR[GP1:91,2] = PR[GP1:90,2] + -16.615;
   1:L PR[91] 10mm/sec CNT100;
   1:  PR[GP1:91,1] = PR[GP1:90,1] + 9.635;
   1:  PR[GP1:91,2] = PR[GP1:90,2] + -17.132;
   1:L PR[91] 10mm/sec CNT100;
   1:  PR[GP1:91,1] = PR[GP1:90,1] + 16.973;
   1:  PR[GP1:91,2] = PR[GP1:90,2] + -25.837;
   1:L PR[91] 10mm/sec CNT100;
   1:  PR[GP1:91,1] = PR[GP1:90,1] + 17.806;
   1:  PR[GP1:91,2] = PR[GP1:90,2] + -26.620;
   1:L PR[91] 10mm/sec CNT100;
   1:  PR[GP1:91,1] = PR[GP1:90,1] + 18.811;
   1:  PR[GP1:91,2] = PR[GP1:90,2] + -27.213;
   1:L PR[91] 10mm/sec CNT100;
   1:  PR[GP1:91,1] = PR[GP1:90,1] + 28.174;
   1:  PR[GP1:91,2] = PR[GP1:90,2] + -32.263;
   1:L PR[91] 10mm/sec CNT100;
   1:  PR[GP1:91,1] = PR[GP1:90,1] + 29.799;
   1:  PR[GP1:91,2] = PR[GP1:90,2] + -32.787;
   1:L PR[91] 10mm/sec CNT100;
   1:  PR[GP1:91,1] = PR[GP1:90,1] + 31.563;
   1:  PR[GP1:91,2] = PR[GP1:90,2] + -32.946;
   1:L PR[91] 10mm/sec CNT100;
   1:  PR[GP1:91,1] = PR[GP1:90,1] + 41.330;
   1:  PR[GP1:91,2] = PR[GP1:90,2] + -34.110;
   1:L PR[91] 10mm/sec CNT100;
   1:  PR[GP1:91,1] = PR[GP1:90,1] + 43.572;
   1:  PR[GP1:91,2] = PR[GP1:90,2] + -33.814;
   1:L PR[91] 10mm/sec CNT100;
   1:  PR[GP1:91,1] = PR[GP1:90,1] + 51.921;
   1:  PR[GP1:91,2] = PR[GP1:90,2] + -31.649;
   1:L PR[91] 10mm/sec CNT100;
   1:  PR[GP1:91,1] = PR[GP1:90,1] + 54.471;
   1:  PR[GP1:91,2] = PR[GP1:90,2] + -30.710;
   1:L PR[91] 10mm/sec CNT100;
   1:  PR[GP1:91,1] = PR[GP1:90,1] + 56.764;
   1:  PR[GP1:91,2] = PR[GP1:90,2] + -29.227;
   1:L PR[91] 10mm/sec CNT100;
   1:  PR[GP1:91,1] = PR[GP1:90,1] + 63.297;
   1:  PR[GP1:91,2] = PR[GP1:90,2] + -24.472;
   1:L PR[91] 10mm/sec CNT100;
   1:  PR[GP1:91,1] = PR[GP1:90,1] + 65.404;
   1:  PR[GP1:91,2] = PR[GP1:90,2] + -22.321;
   1:L PR[91] 10mm/sec CNT100;
   1:  PR[GP1:91,1] = PR[GP1:90,1] + 67.016;
   1:  PR[GP1:91,2] = PR[GP1:90,2] + -19.714;
   1:L PR[91] 10mm/sec CNT100;
   1:  PR[GP1:91,1] = PR[GP1:90,1] + 71.122;
   1:  PR[GP1:91,2] = PR[GP1:90,2] + -13.229;
   1:L PR[91] 10mm/sec CNT100;
   1:  PR[GP1:91,1] = PR[GP1:90,1] + 72.158;
   1:  PR[GP1:91,2] = PR[GP1:90,2] + -10.225;
   1:L PR[91] 10mm/sec CNT100;
   1:  PR[GP1:91,1] = PR[GP1:90,1] + 72.520;
   1:  PR[GP1:91,2] = PR[GP1:90,2] + -6.974;
   1:L PR[91] 10mm/sec CNT100;
   1:  PR[GP1:91,1] = PR[GP1:90,1] + 73.898;
   1:  PR[GP1:91,2] = PR[GP1:90,2] + 0.302;
   1:L PR[91] 10mm/sec CNT100;
   1:  PR[GP1:91,1] = PR[GP1:90,1] + 73.525;
   1:  PR[GP1:91,2] = PR[GP1:90,2] + 3.654;
   1:L PR[91] 10mm/sec CNT100;
   1:  PR[GP1:91,1] = PR[GP1:90,1] + 72.166;
   1:  PR[GP1:91,2] = PR[GP1:90,2] + 10.761;
   1:L PR[91] 10mm/sec CNT100;
   1:  PR[GP1:91,1] = PR[GP1:90,1] + 71.121;
   1:  PR[GP1:91,2] = PR[GP1:90,2] + 13.791;
   1:L PR[91] 10mm/sec CNT100;
   1:  PR[GP1:91,1] = PR[GP1:90,1] + 69.415;
   1:  PR[GP1:91,2] = PR[GP1:90,2] + 16.551;
   1:L PR[91] 10mm/sec CNT100;
   1:  PR[GP1:91,1] = PR[GP1:90,1] + 65.406;
   1:  PR[GP1:91,2] = PR[GP1:90,2] + 22.876;
   1:L PR[91] 10mm/sec CNT100;
   1:  PR[GP1:91,1] = PR[GP1:90,1] + 63.308;
   1:  PR[GP1:91,2] = PR[GP1:90,2] + 25.018;
   1:L PR[91] 10mm/sec CNT100;
   1:  PR[GP1:91,1] = PR[GP1:90,1] + 60.723;
   1:  PR[GP1:91,2] = PR[GP1:90,2] + 26.691;
   1:L PR[91] 10mm/sec CNT100;
   1:  PR[GP1:91,1] = PR[GP1:90,1] + 54.455;
   1:  PR[GP1:91,2] = PR[GP1:90,2] + 31.275;
   1:L PR[91] 10mm/sec CNT100;
   1:  PR[GP1:91,1] = PR[GP1:90,1] + 51.921;
   1:  PR[GP1:91,2] = PR[GP1:90,2] + 32.207;
   1:L PR[91] 10mm/sec CNT100;
   1:  PR[GP1:91,1] = PR[GP1:90,1] + 43.572;
   1:  PR[GP1:91,2] = PR[GP1:90,2] + 34.372;
   1:L PR[91] 10mm/sec CNT100;
   1:  PR[GP1:91,1] = PR[GP1:90,1] + 41.322;
   1:  PR[GP1:91,2] = PR[GP1:90,2] + 34.670;
   1:L PR[91] 10mm/sec CNT100;
   1:  PR[GP1:91,1] = PR[GP1:90,1] + 39.034;
   1:  PR[GP1:91,2] = PR[GP1:90,2] + 34.463;
   1:L PR[91] 10mm/sec CNT100;
   1:  PR[GP1:91,1] = PR[GP1:90,1] + 29.808;
   1:  PR[GP1:91,2] = PR[GP1:90,2] + 33.348;
   1:L PR[91] 10mm/sec CNT100;
   1:  PR[GP1:91,1] = PR[GP1:90,1] + 28.185;
   1:  PR[GP1:91,2] = PR[GP1:90,2] + 32.825;
   1:L PR[91] 10mm/sec CNT100;
   1:  PR[GP1:91,1] = PR[GP1:90,1] + 26.657;
   1:  PR[GP1:91,2] = PR[GP1:90,2] + 31.923;
   1:L PR[91] 10mm/sec CNT100;
   1:  PR[GP1:91,1] = PR[GP1:90,1] + 17.797;
   1:  PR[GP1:91,2] = PR[GP1:90,2] + 27.169;
   1:L PR[91] 10mm/sec CNT100;
   1:  PR[GP1:91,1] = PR[GP1:90,1] + 16.973;
   1:  PR[GP1:91,2] = PR[GP1:90,2] + 26.395;
   1:L PR[91] 10mm/sec CNT100;
   1:  PR[GP1:91,1] = PR[GP1:90,1] + 9.635;
   1:  PR[GP1:91,2] = PR[GP1:90,2] + 17.690;
   1:L PR[91] 10mm/sec CNT100;
   1:  PR[GP1:91,1] = PR[GP1:90,1] + 9.277;
   1:  PR[GP1:91,2] = PR[GP1:90,2] + 17.161;
   1:L PR[91] 10mm/sec CNT100;
   1:  PR[GP1:91,1] = PR[GP1:90,1] + 9.038;
   1:  PR[GP1:91,2] = PR[GP1:90,2] + 16.550;
   1:L PR[91] 10mm/sec CNT100;
   1:  PR[GP1:91,1] = PR[GP1:90,1] + 5.211;
   1:  PR[GP1:91,2] = PR[GP1:90,2] + 5.279;
   1:L PR[91] 10mm/sec CNT100;
   1:  PR[GP1:91,1] = PR[GP1:90,1] + 5.083;
   1:  PR[GP1:91,2] = PR[GP1:90,2] + 4.341;
   1:L PR[91] 10mm/sec CNT100;
   1:  PR[GP1:91,1] = PR[GP1:90,1] + -5.610;
   1:L PR[91] 10mm/sec CNT100;
   1:  PR[GP1:91,1] = PR[GP1:90,1] + -5.736;
   1:  PR[GP1:91,2] = PR[GP1:90,2] + 5.269;
   1:L PR[91] 10mm/sec CNT100;
   1:  PR[GP1:91,1] = PR[GP1:90,1] + -5.885;
   1:  PR[GP1:91,2] = PR[GP1:90,2] + 5.649;
   1:L PR[91] 10mm/sec CNT100;
   1:  PR[GP1:91,1] = PR[GP1:90,1] + -9.815;
   1:  PR[GP1:91,2] = PR[GP1:90,2] + 17.181;
   1:L PR[91] 10mm/sec CNT100;
   1:  PR[GP1:91,1] = PR[GP1:90,1] + -10.165;
   1:  PR[GP1:91,2] = PR[GP1:90,2] + 17.699;
   1:L PR[91] 10mm/sec CNT100;
   1:  PR[GP1:91,1] = PR[GP1:90,1] + -17.503;
   1:  PR[GP1:91,2] = PR[GP1:90,2] + 26.397;
   1:L PR[91] 10mm/sec CNT100;
   1:  PR[GP1:91,1] = PR[GP1:90,1] + -18.336;
   1:  PR[GP1:91,2] = PR[GP1:90,2] + 27.180;
   1:L PR[91] 10mm/sec CNT100;
   1:  PR[GP1:91,1] = PR[GP1:90,1] + -19.341;
   1:  PR[GP1:91,2] = PR[GP1:90,2] + 27.773;
   1:L PR[91] 10mm/sec CNT100;
   1:  PR[GP1:91,1] = PR[GP1:90,1] + -28.704;
   1:  PR[GP1:91,2] = PR[GP1:90,2] + 32.823;
   1:L PR[91] 10mm/sec CNT100;
   1:  PR[GP1:91,1] = PR[GP1:90,1] + -30.330;
   1:  PR[GP1:91,2] = PR[GP1:90,2] + 33.347;
   1:L PR[91] 10mm/sec CNT100;
   1:  PR[GP1:91,1] = PR[GP1:90,1] + -32.094;
   1:  PR[GP1:91,2] = PR[GP1:90,2] + 33.506;
   1:L PR[91] 10mm/sec CNT100;
   1:  PR[GP1:91,1] = PR[GP1:90,1] + -41.860;
   1:  PR[GP1:91,2] = PR[GP1:90,2] + 34.668;
   1:L PR[91] 10mm/sec CNT100;
   1:  PR[GP1:91,1] = PR[GP1:90,1] + -44.101;
   1:  PR[GP1:91,2] = PR[GP1:90,2] + 34.372;
   1:L PR[91] 10mm/sec CNT100;
   1:  PR[GP1:91,1] = PR[GP1:90,1] + -52.450;
   1:  PR[GP1:91,2] = PR[GP1:90,2] + 32.207;
   1:L PR[91] 10mm/sec CNT100;
   1:  PR[GP1:91,1] = PR[GP1:90,1] + -55.000;
   1:  PR[GP1:91,2] = PR[GP1:90,2] + 31.268;
   1:L PR[91] 10mm/sec CNT100;
   1:  PR[GP1:91,1] = PR[GP1:90,1] + -57.292;
   1:  PR[GP1:91,2] = PR[GP1:90,2] + 29.785;
   1:L PR[91] 10mm/sec CNT100;
   1:  PR[GP1:91,1] = PR[GP1:90,1] + -63.824;
   1:  PR[GP1:91,2] = PR[GP1:90,2] + 25.030;
   1:L PR[91] 10mm/sec CNT100;
   1:  PR[GP1:91,1] = PR[GP1:90,1] + -65.931;
   1:  PR[GP1:91,2] = PR[GP1:90,2] + 22.878;
   1:L PR[91] 10mm/sec CNT100;
   1:  PR[GP1:91,1] = PR[GP1:90,1] + -67.543;
   1:  PR[GP1:91,2] = PR[GP1:90,2] + 20.271;
   1:L PR[91] 10mm/sec CNT100;
   1:  PR[GP1:91,1] = PR[GP1:90,1] + -71.649;
   1:  PR[GP1:91,2] = PR[GP1:90,2] + 13.785;
   1:L PR[91] 10mm/sec CNT100;
   1:  PR[GP1:91,1] = PR[GP1:90,1] + -72.685;
   1:  PR[GP1:91,2] = PR[GP1:90,2] + 10.781;
   1:L PR[91] 10mm/sec CNT100;
   1:  PR[GP1:91,1] = PR[GP1:90,1] + -73.047;
   1:  PR[GP1:91,2] = PR[GP1:90,2] + 7.530;
   1:L PR[91] 10mm/sec CNT100;
   1:  PR[GP1:91,1] = PR[GP1:90,1] + -74.424;
   1:  PR[GP1:91,2] = PR[GP1:90,2] + 0.256;
   1:L PR[91] 10mm/sec CNT100;
   1:  PR[GP1:91,1] = PR[GP1:90,1] + -74.052;
   1:  PR[GP1:91,2] = PR[GP1:90,2] + -3.096;
   1:L PR[91] 10mm/sec CNT100;
   1:  PR[GP1:91,1] = PR[GP1:90,1] + -72.693;
   1:  PR[GP1:91,2] = PR[GP1:90,2] + -10.200;
   1:L PR[91] 10mm/sec CNT100;
   1:  PR[GP1:91,1] = PR[GP1:90,1] + -71.648;
   1:  PR[GP1:91,2] = PR[GP1:90,2] + -13.230;
   1:L PR[91] 10mm/sec CNT100;
   1:  PR[GP1:91,1] = PR[GP1:90,1] + -69.942;
   1:  PR[GP1:91,2] = PR[GP1:90,2] + -15.990;
   1:L PR[91] 10mm/sec CNT100;
   1:  PR[GP1:91,1] = PR[GP1:90,1] + -65.934;
   1:  PR[GP1:91,2] = PR[GP1:90,2] + -22.318;
   1:L PR[91] 10mm/sec CNT100;
   1:  PR[GP1:91,1] = PR[GP1:90,1] + -63.835;
   1:  PR[GP1:91,2] = PR[GP1:90,2] + -24.460;
   1:L PR[91] 10mm/sec CNT100;
   1:  PR[GP1:91,1] = PR[GP1:90,1] + -61.250;
   1:  PR[GP1:91,2] = PR[GP1:90,2] + -26.132;
   1:L PR[91] 10mm/sec CNT100;
   1:  PR[GP1:91,1] = PR[GP1:90,1] + -54.983;
   1:  PR[GP1:91,2] = PR[GP1:90,2] + -30.716;
   1:L PR[91] 10mm/sec CNT100;
   1:  PR[GP1:91,1] = PR[GP1:90,1] + -52.450;
   1:  PR[GP1:91,2] = PR[GP1:90,2] + -31.648;
   1:L PR[91] 10mm/sec CNT100;
   1:  PR[GP1:91,1] = PR[GP1:90,1] + -44.101;
   1:  PR[GP1:91,2] = PR[GP1:90,2] + -33.814;
   1:L PR[91] 10mm/sec CNT100;
   1:  PR[GP1:91,1] = PR[GP1:90,1] + -41.851;
   1:  PR[GP1:91,2] = PR[GP1:90,2] + -34.111;
   1:L PR[91] 10mm/sec CNT100;
   1:  PR[GP1:91,1] = PR[GP1:90,1] + -39.563;
   1:  PR[GP1:91,2] = PR[GP1:90,2] + -33.905;
   1:L PR[91] 10mm/sec CNT100;
   1:  PR[GP1:91,1] = PR[GP1:90,1] + -30.338;
   1:  PR[GP1:91,2] = PR[GP1:90,2] + -32.791;
   1:L PR[91] 10mm/sec CNT100;
   1:  PR[GP1:91,1] = PR[GP1:90,1] + -28.715;
   1:  PR[GP1:91,2] = PR[GP1:90,2] + -32.269;
   1:L PR[91] 10mm/sec CNT100;
   1:  PR[GP1:91,1] = PR[GP1:90,1] + -27.187;
   1:  PR[GP1:91,2] = PR[GP1:90,2] + -31.367;
   1:L PR[91] 10mm/sec CNT100;
   1:  PR[GP1:91,1] = PR[GP1:90,1] + -18.327;
   1:  PR[GP1:91,2] = PR[GP1:90,2] + -26.614;
   1:L PR[91] 10mm/sec CNT100;
   1:  PR[GP1:91,1] = PR[GP1:90,1] + -17.503;
   1:  PR[GP1:91,2] = PR[GP1:90,2] + -25.839;
   1:L PR[91] 10mm/sec CNT100;
   1:  PR[GP1:91,1] = PR[GP1:90,1] + -10.165;
   1:  PR[GP1:91,2] = PR[GP1:90,2] + -17.141;
   1:L PR[91] 10mm/sec CNT100;
   1:  PR[GP1:91,1] = PR[GP1:90,1] + -9.807;
   1:  PR[GP1:91,2] = PR[GP1:90,2] + -16.611;
   1:L PR[91] 10mm/sec CNT100;
   1:  PR[GP1:91,1] = PR[GP1:90,1] + -9.567;
   1:  PR[GP1:91,2] = PR[GP1:90,2] + -15.999;
   1:L PR[91] 10mm/sec CNT100;
   1:  PR[GP1:91,1] = PR[GP1:90,1] + -5.737;
   1:  PR[GP1:91,2] = PR[GP1:90,2] + -4.721;
   1:L PR[91] 10mm/sec CNT100;
   1:  PR[GP1:91,1] = PR[GP1:90,1] + -5.610;
   1:  PR[GP1:91,2] = PR[GP1:90,2] + -3.783;
   1:L PR[91] 10mm/sec CNT100;
   1:  PR[GP1:91,1] = PR[GP1:90,1] + 5.083;
   1:L PR[91] 10mm/sec CNT100;
   1:  PR[GP1:91,1] = PR[GP1:90,1] + 7.931;
   1:  PR[GP1:91,2] = PR[GP1:90,2] + -12.727;
   1:  PR[GP1:91,3] = PR[GP1:90,3] + 15.555;
   1:L PR[91] 10mm/sec CNT100;
   1:  PR[GP1:91,1] = PR[GP1:90,1] + 9.273;
   1:  PR[GP1:91,2] = PR[GP1:90,2] + -16.664;
   1:L PR[91] 10mm/sec CNT100;
   1:  PR[GP1:91,1] = PR[GP1:90,1] + 17.289;
   1:  PR[GP1:91,2] = PR[GP1:90,2] + -26.189;
   1:L PR[91] 10mm/sec CNT100;
   1:  PR[GP1:91,1] = PR[GP1:90,1] + 17.688;
   1:  PR[GP1:91,2] = PR[GP1:90,2] + -26.564;
   1:L PR[91] 10mm/sec CNT100;
   1:  PR[GP1:91,1] = PR[GP1:90,1] + 18.179;
   1:  PR[GP1:91,2] = PR[GP1:90,2] + -26.853;
   1:L PR[91] 10mm/sec CNT100;
   1:  PR[GP1:91,1] = PR[GP1:90,1] + 28.408;
   1:  PR[GP1:91,2] = PR[GP1:90,2] + -32.371;
   1:L PR[91] 10mm/sec CNT100;
   1:  PR[GP1:91,1] = PR[GP1:90,1] + 29.517;
   1:  PR[GP1:91,2] = PR[GP1:90,2] + -32.728;
   1:L PR[91] 10mm/sec CNT100;
   1:  PR[GP1:91,1] = PR[GP1:90,1] + 30.740;
   1:  PR[GP1:91,2] = PR[GP1:90,2] + -32.839;
   1:L PR[91] 10mm/sec CNT100;
   1:  PR[GP1:91,1] = PR[GP1:90,1] + 41.411;
   1:  PR[GP1:91,2] = PR[GP1:90,2] + -34.111;
   1:L PR[91] 10mm/sec CNT100;
   1:  PR[GP1:91,1] = PR[GP1:90,1] + 43.164;
   1:  PR[GP1:91,2] = PR[GP1:90,2] + -33.879;
   1:L PR[91] 10mm/sec CNT100;
   1:  PR[GP1:91,1] = PR[GP1:90,1] + 52.287;
   1:  PR[GP1:91,2] = PR[GP1:90,2] + -31.514;
   1:L PR[91] 10mm/sec CNT100;
   1:  PR[GP1:91,1] = PR[GP1:90,1] + 54.412;
   1:  PR[GP1:91,2] = PR[GP1:90,2] + -30.731;
   1:L PR[91] 10mm/sec CNT100;
   1:  PR[GP1:91,1] = PR[GP1:90,1] + 56.325;
   1:  PR[GP1:91,2] = PR[GP1:90,2] + -29.493;
   1:L PR[91] 10mm/sec CNT100;
   1:  PR[GP1:91,1] = PR[GP1:90,1] + 63.463;
   1:  PR[GP1:91,2] = PR[GP1:90,2] + -24.298;
   1:L PR[91] 10mm/sec CNT100;
   1:  PR[GP1:91,1] = PR[GP1:90,1] + 65.274;
   1:  PR[GP1:91,2] = PR[GP1:90,2] + -22.449;
   1:L PR[91] 10mm/sec CNT100;
   1:  PR[GP1:91,1] = PR[GP1:90,1] + 66.663;
   1:  PR[GP1:91,2] = PR[GP1:90,2] + -20.201;
   1:L PR[91] 10mm/sec CNT100;
   1:  PR[GP1:91,1] = PR[GP1:90,1] + 71.150;
   1:  PR[GP1:91,2] = PR[GP1:90,2] + -13.116;
   1:L PR[91] 10mm/sec CNT100;
   1:  PR[GP1:91,1] = PR[GP1:90,1] + 72.054;
   1:  PR[GP1:91,2] = PR[GP1:90,2] + -10.496;
   1:L PR[91] 10mm/sec CNT100;
   1:  PR[GP1:91,1] = PR[GP1:90,1] + 72.371;
   1:  PR[GP1:91,2] = PR[GP1:90,2] + -7.648;
   1:L PR[91] 10mm/sec CNT100;
   1:  PR[GP1:91,1] = PR[GP1:90,1] + 73.877;
   1:  PR[GP1:91,2] = PR[GP1:90,2] + 0.302;
   1:L PR[91] 10mm/sec CNT100;
   1:  PR[GP1:91,1] = PR[GP1:90,1] + 73.547;
   1:  PR[GP1:91,2] = PR[GP1:90,2] + 3.266;
   1:L PR[91] 10mm/sec CNT100;
   1:  PR[GP1:91,1] = PR[GP1:90,1] + 72.062;
   1:  PR[GP1:91,2] = PR[GP1:90,2] + 11.031;
   1:L PR[91] 10mm/sec CNT100;
   1:  PR[GP1:91,1] = PR[GP1:90,1] + 71.149;
   1:  PR[GP1:91,2] = PR[GP1:90,2] + 13.678;
   1:L PR[91] 10mm/sec CNT100;
   1:  PR[GP1:91,1] = PR[GP1:90,1] + 69.657;
   1:  PR[GP1:91,2] = PR[GP1:90,2] + 16.092;
   1:L PR[91] 10mm/sec CNT100;
   1:  PR[GP1:91,1] = PR[GP1:90,1] + 65.277;
   1:  PR[GP1:91,2] = PR[GP1:90,2] + 23.004;
   1:L PR[91] 10mm/sec CNT100;
   1:  PR[GP1:91,1] = PR[GP1:90,1] + 63.475;
   1:  PR[GP1:91,2] = PR[GP1:90,2] + 24.844;
   1:L PR[91] 10mm/sec CNT100;
   1:  PR[GP1:91,1] = PR[GP1:90,1] + 61.245;
   1:  PR[GP1:91,2] = PR[GP1:90,2] + 26.286;
   1:L PR[91] 10mm/sec CNT100;
   1:  PR[GP1:91,1] = PR[GP1:90,1] + 54.396;
   1:  PR[GP1:91,2] = PR[GP1:90,2] + 31.295;
   1:L PR[91] 10mm/sec CNT100;
   1:  PR[GP1:91,1] = PR[GP1:90,1] + 52.287;
   1:  PR[GP1:91,2] = PR[GP1:90,2] + 32.072;
   1:L PR[91] 10mm/sec CNT100;
   1:  PR[GP1:91,1] = PR[GP1:90,1] + 43.164;
   1:  PR[GP1:91,2] = PR[GP1:90,2] + 34.437;
   1:L PR[91] 10mm/sec CNT100;
   1:  PR[GP1:91,1] = PR[GP1:90,1] + 41.402;
   1:  PR[GP1:91,2] = PR[GP1:90,2] + 34.670;
   1:L PR[91] 10mm/sec CNT100;
   1:  PR[GP1:91,1] = PR[GP1:90,1] + 39.605;
   1:  PR[GP1:91,2] = PR[GP1:90,2] + 34.507;
   1:L PR[91] 10mm/sec CNT100;
   1:  PR[GP1:91,1] = PR[GP1:90,1] + 29.526;
   1:  PR[GP1:91,2] = PR[GP1:90,2] + 33.289;
   1:L PR[91] 10mm/sec CNT100;
   1:  PR[GP1:91,1] = PR[GP1:90,1] + 28.419;
   1:  PR[GP1:91,2] = PR[GP1:90,2] + 32.933;
   1:L PR[91] 10mm/sec CNT100;
   1:  PR[GP1:91,1] = PR[GP1:90,1] + 27.358;
   1:  PR[GP1:91,2] = PR[GP1:90,2] + 32.307;
   1:L PR[91] 10mm/sec CNT100;
   1:  PR[GP1:91,1] = PR[GP1:90,1] + 17.679;
   1:  PR[GP1:91,2] = PR[GP1:90,2] + 27.113;
   1:L PR[91] 10mm/sec CNT100;
   1:  PR[GP1:91,1] = PR[GP1:90,1] + 17.289;
   1:  PR[GP1:91,2] = PR[GP1:90,2] + 26.747;
   1:L PR[91] 10mm/sec CNT100;
   1:  PR[GP1:91,1] = PR[GP1:90,1] + 9.273;
   1:  PR[GP1:91,2] = PR[GP1:90,2] + 17.222;
   1:L PR[91] 10mm/sec CNT100;
   1:  PR[GP1:91,1] = PR[GP1:90,1] + 7.952;
   1:  PR[GP1:91,2] = PR[GP1:90,2] + 13.344;
   1:L PR[91] 10mm/sec CNT100;
   1:  PR[GP1:91,1] = PR[GP1:90,1] + 4.948;
   1:  PR[GP1:91,2] = PR[GP1:90,2] + 4.666;
   1:L PR[91] 10mm/sec CNT100;
   1:  PR[GP1:91,1] = PR[GP1:90,1] + -5.475;
   1:L PR[91] 10mm/sec CNT100;
   1:  PR[GP1:91,1] = PR[GP1:90,1] + -8.460;
   1:  PR[GP1:91,2] = PR[GP1:90,2] + 13.291;
   1:L PR[91] 10mm/sec CNT100;
   1:  PR[GP1:91,1] = PR[GP1:90,1] + -9.803;
   1:  PR[GP1:91,2] = PR[GP1:90,2] + 17.231;
   1:L PR[91] 10mm/sec CNT100;
   1:  PR[GP1:91,1] = PR[GP1:90,1] + -17.820;
   1:  PR[GP1:91,2] = PR[GP1:90,2] + 26.750;
   1:L PR[91] 10mm/sec CNT100;
   1:  PR[GP1:91,1] = PR[GP1:90,1] + -18.219;
   1:  PR[GP1:91,2] = PR[GP1:90,2] + 27.124;
   1:L PR[91] 10mm/sec CNT100;
   1:  PR[GP1:91,1] = PR[GP1:90,1] + -18.710;
   1:  PR[GP1:91,2] = PR[GP1:90,2] + 27.415;
   1:L PR[91] 10mm/sec CNT100;
   1:  PR[GP1:91,1] = PR[GP1:90,1] + -28.939;
   1:  PR[GP1:91,2] = PR[GP1:90,2] + 32.931;
   1:L PR[91] 10mm/sec CNT100;
   1:  PR[GP1:91,1] = PR[GP1:90,1] + -30.048;
   1:  PR[GP1:91,2] = PR[GP1:90,2] + 33.288;
   1:L PR[91] 10mm/sec CNT100;
   1:  PR[GP1:91,1] = PR[GP1:90,1] + -31.271;
   1:  PR[GP1:91,2] = PR[GP1:90,2] + 33.399;
   1:L PR[91] 10mm/sec CNT100;
   1:  PR[GP1:91,1] = PR[GP1:90,1] + -41.940;
   1:  PR[GP1:91,2] = PR[GP1:90,2] + 34.668;
   1:L PR[91] 10mm/sec CNT100;
   1:  PR[GP1:91,1] = PR[GP1:90,1] + -43.694;
   1:  PR[GP1:91,2] = PR[GP1:90,2] + 34.437;
   1:L PR[91] 10mm/sec CNT100;
   1:  PR[GP1:91,1] = PR[GP1:90,1] + -52.815;
   1:  PR[GP1:91,2] = PR[GP1:90,2] + 32.071;
   1:L PR[91] 10mm/sec CNT100;
   1:  PR[GP1:91,1] = PR[GP1:90,1] + -54.941;
   1:  PR[GP1:91,2] = PR[GP1:90,2] + 31.288;
   1:L PR[91] 10mm/sec CNT100;
   1:  PR[GP1:91,1] = PR[GP1:90,1] + -56.853;
   1:  PR[GP1:91,2] = PR[GP1:90,2] + 30.051;
   1:L PR[91] 10mm/sec CNT100;
   1:  PR[GP1:91,1] = PR[GP1:90,1] + -63.990;
   1:  PR[GP1:91,2] = PR[GP1:90,2] + 24.855;
   1:L PR[91] 10mm/sec CNT100;
   1:  PR[GP1:91,1] = PR[GP1:90,1] + -65.802;
   1:  PR[GP1:91,2] = PR[GP1:90,2] + 23.006;
   1:L PR[91] 10mm/sec CNT100;
   1:  PR[GP1:91,1] = PR[GP1:90,1] + -67.191;
   1:  PR[GP1:91,2] = PR[GP1:90,2] + 20.759;
   1:L PR[91] 10mm/sec CNT100;
   1:  PR[GP1:91,1] = PR[GP1:90,1] + -71.677;
   1:  PR[GP1:91,2] = PR[GP1:90,2] + 13.672;
   1:L PR[91] 10mm/sec CNT100;
   1:  PR[GP1:91,1] = PR[GP1:90,1] + -72.581;
   1:  PR[GP1:91,2] = PR[GP1:90,2] + 11.052;
   1:L PR[91] 10mm/sec CNT100;
   1:  PR[GP1:91,1] = PR[GP1:90,1] + -72.897;
   1:  PR[GP1:91,2] = PR[GP1:90,2] + 8.204;
   1:L PR[91] 10mm/sec CNT100;
   1:  PR[GP1:91,1] = PR[GP1:90,1] + -74.403;
   1:  PR[GP1:91,2] = PR[GP1:90,2] + 0.256;
   1:L PR[91] 10mm/sec CNT100;
   1:  PR[GP1:91,1] = PR[GP1:90,1] + -74.073;
   1:  PR[GP1:91,2] = PR[GP1:90,2] + -2.708;
   1:L PR[91] 10mm/sec CNT100;
   1:  PR[GP1:91,1] = PR[GP1:90,1] + -72.589;
   1:  PR[GP1:91,2] = PR[GP1:90,2] + -10.471;
   1:L PR[91] 10mm/sec CNT100;
   1:  PR[GP1:91,1] = PR[GP1:90,1] + -71.676;
   1:  PR[GP1:91,2] = PR[GP1:90,2] + -13.117;
   1:L PR[91] 10mm/sec CNT100;
   1:  PR[GP1:91,1] = PR[GP1:90,1] + -70.183;
   1:  PR[GP1:91,2] = PR[GP1:90,2] + -15.532;
   1:L PR[91] 10mm/sec CNT100;
   1:  PR[GP1:91,1] = PR[GP1:90,1] + -65.804;
   1:  PR[GP1:91,2] = PR[GP1:90,2] + -22.446;
   1:L PR[91] 10mm/sec CNT100;
   1:  PR[GP1:91,1] = PR[GP1:90,1] + -64.002;
   1:  PR[GP1:91,2] = PR[GP1:90,2] + -24.285;
   1:L PR[91] 10mm/sec CNT100;
   1:  PR[GP1:91,1] = PR[GP1:90,1] + -61.772;
   1:  PR[GP1:91,2] = PR[GP1:90,2] + -25.728;
   1:L PR[91] 10mm/sec CNT100;
   1:  PR[GP1:91,1] = PR[GP1:90,1] + -54.924;
   1:  PR[GP1:91,2] = PR[GP1:90,2] + -30.736;
   1:L PR[91] 10mm/sec CNT100;
   1:  PR[GP1:91,1] = PR[GP1:90,1] + -52.815;
   1:  PR[GP1:91,2] = PR[GP1:90,2] + -31.513;
   1:L PR[91] 10mm/sec CNT100;
   1:  PR[GP1:91,1] = PR[GP1:90,1] + -43.694;
   1:  PR[GP1:91,2] = PR[GP1:90,2] + -33.879;
   1:L PR[91] 10mm/sec CNT100;
   1:  PR[GP1:91,1] = PR[GP1:90,1] + -41.932;
   1:  PR[GP1:91,2] = PR[GP1:90,2] + -34.111;
   1:L PR[91] 10mm/sec CNT100;
   1:  PR[GP1:91,1] = PR[GP1:90,1] + -40.135;
   1:  PR[GP1:91,2] = PR[GP1:90,2] + -33.949;
   1:L PR[91] 10mm/sec CNT100;
   1:  PR[GP1:91,1] = PR[GP1:90,1] + -30.056;
   1:  PR[GP1:91,2] = PR[GP1:90,2] + -32.733;
   1:L PR[91] 10mm/sec CNT100;
   1:  PR[GP1:91,1] = PR[GP1:90,1] + -28.950;
   1:  PR[GP1:91,2] = PR[GP1:90,2] + -32.376;
   1:L PR[91] 10mm/sec CNT100;
   1:  PR[GP1:91,1] = PR[GP1:90,1] + -27.889;
   1:  PR[GP1:91,2] = PR[GP1:90,2] + -31.750;
   1:L PR[91] 10mm/sec CNT100;
   1:  PR[GP1:91,1] = PR[GP1:90,1] + -18.210;
   1:  PR[GP1:91,2] = PR[GP1:90,2] + -26.558;
   1:L PR[91] 10mm/sec CNT100;
   1:  PR[GP1:91,1] = PR[GP1:90,1] + -17.820;
   1:  PR[GP1:91,2] = PR[GP1:90,2] + -26.192;
   1:L PR[91] 10mm/sec CNT100;
   1:  PR[GP1:91,1] = PR[GP1:90,1] + -9.803;
   1:  PR[GP1:91,2] = PR[GP1:90,2] + -16.673;
   1:L PR[91] 10mm/sec CNT100;
   1:  PR[GP1:91,1] = PR[GP1:90,1] + -8.481;
   1:  PR[GP1:91,2] = PR[GP1:90,2] + -12.791;
   1:L PR[91] 10mm/sec CNT100;
   1:  PR[GP1:91,1] = PR[GP1:90,1] + -5.474;
   1:  PR[GP1:91,2] = PR[GP1:90,2] + -4.108;
   1:L PR[91] 10mm/sec CNT100;
   1:  PR[GP1:91,1] = PR[GP1:90,1] + 4.948;
   1:L PR[91] 10mm/sec CNT100;
   1:  PR[GP1:91,1] = PR[GP1:90,1] + 8.918;
   1:  PR[GP1:91,2] = PR[GP1:90,2] + -16.091;
   1:  PR[GP1:91,3] = PR[GP1:90,3] + 16.165;
   1:L PR[91] 10mm/sec CNT100;
   1:  PR[GP1:91,1] = PR[GP1:90,1] + 9.271;
   1:  PR[GP1:91,2] = PR[GP1:90,2] + -16.852;
   1:L PR[91] 10mm/sec CNT100;
   1:  PR[GP1:91,1] = PR[GP1:90,1] + 17.590;
   1:  PR[GP1:91,2] = PR[GP1:90,2] + -26.515;
   1:L PR[91] 10mm/sec CNT100;
   1:  PR[GP1:91,1] = PR[GP1:90,1] + 28.642;
   1:  PR[GP1:91,2] = PR[GP1:90,2] + -32.479;
   1:L PR[91] 10mm/sec CNT100;
   1:  PR[GP1:91,1] = PR[GP1:90,1] + 29.234;
   1:  PR[GP1:91,2] = PR[GP1:90,2] + -32.669;
   1:L PR[91] 10mm/sec CNT100;
   1:  PR[GP1:91,1] = PR[GP1:90,1] + 29.917;
   1:  PR[GP1:91,2] = PR[GP1:90,2] + -32.731;
   1:L PR[91] 10mm/sec CNT100;
   1:  PR[GP1:91,1] = PR[GP1:90,1] + 41.491;
   1:  PR[GP1:91,2] = PR[GP1:90,2] + -34.111;
   1:L PR[91] 10mm/sec CNT100;
   1:  PR[GP1:91,1] = PR[GP1:90,1] + 42.756;
   1:  PR[GP1:91,2] = PR[GP1:90,2] + -33.944;
   1:L PR[91] 10mm/sec CNT100;
   1:  PR[GP1:91,1] = PR[GP1:90,1] + 52.652;
   1:  PR[GP1:91,2] = PR[GP1:90,2] + -31.378;
   1:L PR[91] 10mm/sec CNT100;
   1:  PR[GP1:91,1] = PR[GP1:90,1] + 54.353;
   1:  PR[GP1:91,2] = PR[GP1:90,2] + -30.751;
   1:L PR[91] 10mm/sec CNT100;
   1:  PR[GP1:91,1] = PR[GP1:90,1] + 55.886;
   1:  PR[GP1:91,2] = PR[GP1:90,2] + -29.759;
   1:L PR[91] 10mm/sec CNT100;
   1:  PR[GP1:91,1] = PR[GP1:90,1] + 63.629;
   1:  PR[GP1:91,2] = PR[GP1:90,2] + -24.123;
   1:L PR[91] 10mm/sec CNT100;
   1:  PR[GP1:91,1] = PR[GP1:90,1] + 65.144;
   1:  PR[GP1:91,2] = PR[GP1:90,2] + -22.577;
   1:L PR[91] 10mm/sec CNT100;
   1:  PR[GP1:91,1] = PR[GP1:90,1] + 66.311;
   1:  PR[GP1:91,2] = PR[GP1:90,2] + -20.689;
   1:L PR[91] 10mm/sec CNT100;
   1:  PR[GP1:91,1] = PR[GP1:90,1] + 71.178;
   1:  PR[GP1:91,2] = PR[GP1:90,2] + -13.003;
   1:L PR[91] 10mm/sec CNT100;
   1:  PR[GP1:91,1] = PR[GP1:90,1] + 71.950;
   1:  PR[GP1:91,2] = PR[GP1:90,2] + -10.767;
   1:L PR[91] 10mm/sec CNT100;
   1:  PR[GP1:91,1] = PR[GP1:90,1] + 72.222;
   1:  PR[GP1:91,2] = PR[GP1:90,2] + -8.323;
   1:L PR[91] 10mm/sec CNT100;
   1:  PR[GP1:91,1] = PR[GP1:90,1] + 73.855;
   1:  PR[GP1:91,2] = PR[GP1:90,2] + 0.302;
   1:L PR[91] 10mm/sec CNT100;
   1:  PR[GP1:91,1] = PR[GP1:90,1] + 73.569;
   1:  PR[GP1:91,2] = PR[GP1:90,2] + 2.879;
   1:L PR[91] 10mm/sec CNT100;
   1:  PR[GP1:91,1] = PR[GP1:90,1] + 71.958;
   1:  PR[GP1:91,2] = PR[GP1:90,2] + 11.302;
   1:L PR[91] 10mm/sec CNT100;
   1:  PR[GP1:91,1] = PR[GP1:90,1] + 71.177;
   1:  PR[GP1:91,2] = PR[GP1:90,2] + 13.565;
   1:L PR[91] 10mm/sec CNT100;
   1:  PR[GP1:91,1] = PR[GP1:90,1] + 69.898;
   1:  PR[GP1:91,2] = PR[GP1:90,2] + 15.634;
   1:L PR[91] 10mm/sec CNT100;
   1:  PR[GP1:91,1] = PR[GP1:90,1] + 65.147;
   1:  PR[GP1:91,2] = PR[GP1:90,2] + 23.132;
   1:L PR[91] 10mm/sec CNT100;
   1:  PR[GP1:91,1] = PR[GP1:90,1] + 63.641;
   1:  PR[GP1:91,2] = PR[GP1:90,2] + 24.669;
   1:L PR[91] 10mm/sec CNT100;
   1:  PR[GP1:91,1] = PR[GP1:90,1] + 61.767;
   1:  PR[GP1:91,2] = PR[GP1:90,2] + 25.882;
   1:L PR[91] 10mm/sec CNT100;
   1:  PR[GP1:91,1] = PR[GP1:90,1] + 54.337;
   1:  PR[GP1:91,2] = PR[GP1:90,2] + 31.315;
   1:L PR[91] 10mm/sec CNT100;
   1:  PR[GP1:91,1] = PR[GP1:90,1] + 52.652;
   1:  PR[GP1:91,2] = PR[GP1:90,2] + 31.936;
   1:L PR[91] 10mm/sec CNT100;
   1:  PR[GP1:91,1] = PR[GP1:90,1] + 42.756;
   1:  PR[GP1:91,2] = PR[GP1:90,2] + 34.502;
   1:L PR[91] 10mm/sec CNT100;
   1:  PR[GP1:91,1] = PR[GP1:90,1] + 41.483;
   1:  PR[GP1:91,2] = PR[GP1:90,2] + 34.670;
   1:L PR[91] 10mm/sec CNT100;
   1:  PR[GP1:91,1] = PR[GP1:90,1] + 40.176;
   1:  PR[GP1:91,2] = PR[GP1:90,2] + 34.552;
   1:L PR[91] 10mm/sec CNT100;
   1:  PR[GP1:91,1] = PR[GP1:90,1] + 29.243;
   1:  PR[GP1:91,2] = PR[GP1:90,2] + 33.230;
   1:L PR[91] 10mm/sec CNT100;
   1:  PR[GP1:91,1] = PR[GP1:90,1] + 28.653;
   1:  PR[GP1:91,2] = PR[GP1:90,2] + 33.040;
   1:L PR[91] 10mm/sec CNT100;
   1:  PR[GP1:91,1] = PR[GP1:90,1] + 28.060;
   1:  PR[GP1:91,2] = PR[GP1:90,2] + 32.690;
   1:L PR[91] 10mm/sec CNT100;
   1:  PR[GP1:91,1] = PR[GP1:90,1] + 17.589;
   1:  PR[GP1:91,2] = PR[GP1:90,2] + 27.072;
   1:L PR[91] 10mm/sec CNT100;
   1:  PR[GP1:91,1] = PR[GP1:90,1] + 9.271;
   1:  PR[GP1:91,2] = PR[GP1:90,2] + 17.409;
   1:L PR[91] 10mm/sec CNT100;
   1:  PR[GP1:91,1] = PR[GP1:90,1] + 8.918;
   1:  PR[GP1:91,2] = PR[GP1:90,2] + 16.648;
   1:L PR[91] 10mm/sec CNT100;
   1:  PR[GP1:91,1] = PR[GP1:90,1] + 4.882;
   1:  PR[GP1:91,2] = PR[GP1:90,2] + 4.991;
   1:L PR[91] 10mm/sec CNT100;
   1:  PR[GP1:91,1] = PR[GP1:90,1] + -5.409;
   1:L PR[91] 10mm/sec CNT100;
   1:  PR[GP1:91,1] = PR[GP1:90,1] + -9.448;
   1:  PR[GP1:91,2] = PR[GP1:90,2] + 16.658;
   1:L PR[91] 10mm/sec CNT100;
   1:  PR[GP1:91,1] = PR[GP1:90,1] + -9.802;
   1:  PR[GP1:91,2] = PR[GP1:90,2] + 17.420;
   1:L PR[91] 10mm/sec CNT100;
   1:  PR[GP1:91,1] = PR[GP1:90,1] + -18.121;
   1:  PR[GP1:91,2] = PR[GP1:90,2] + 27.076;
   1:L PR[91] 10mm/sec CNT100;
   1:  PR[GP1:91,1] = PR[GP1:90,1] + -29.173;
   1:  PR[GP1:91,2] = PR[GP1:90,2] + 33.039;
   1:L PR[91] 10mm/sec CNT100;
   1:  PR[GP1:91,1] = PR[GP1:90,1] + -29.765;
   1:  PR[GP1:91,2] = PR[GP1:90,2] + 33.229;
   1:L PR[91] 10mm/sec CNT100;
   1:  PR[GP1:91,1] = PR[GP1:90,1] + -30.449;
   1:  PR[GP1:91,2] = PR[GP1:90,2] + 33.291;
   1:L PR[91] 10mm/sec CNT100;
   1:  PR[GP1:91,1] = PR[GP1:90,1] + -42.021;
   1:  PR[GP1:91,2] = PR[GP1:90,2] + 34.668;
   1:L PR[91] 10mm/sec CNT100;
   1:  PR[GP1:91,1] = PR[GP1:90,1] + -43.286;
   1:  PR[GP1:91,2] = PR[GP1:90,2] + 34.501;
   1:L PR[91] 10mm/sec CNT100;
   1:  PR[GP1:91,1] = PR[GP1:90,1] + -53.180;
   1:  PR[GP1:91,2] = PR[GP1:90,2] + 31.935;
   1:L PR[91] 10mm/sec CNT100;
   1:  PR[GP1:91,1] = PR[GP1:90,1] + -54.882;
   1:  PR[GP1:91,2] = PR[GP1:90,2] + 31.308;
   1:L PR[91] 10mm/sec CNT100;
   1:  PR[GP1:91,1] = PR[GP1:90,1] + -56.415;
   1:  PR[GP1:91,2] = PR[GP1:90,2] + 30.316;
   1:L PR[91] 10mm/sec CNT100;
   1:  PR[GP1:91,1] = PR[GP1:90,1] + -64.157;
   1:  PR[GP1:91,2] = PR[GP1:90,2] + 24.681;
   1:L PR[91] 10mm/sec CNT100;
   1:  PR[GP1:91,1] = PR[GP1:90,1] + -65.672;
   1:  PR[GP1:91,2] = PR[GP1:90,2] + 23.134;
   1:L PR[91] 10mm/sec CNT100;
   1:  PR[GP1:91,1] = PR[GP1:90,1] + -66.838;
   1:  PR[GP1:91,2] = PR[GP1:90,2] + 21.247;
   1:L PR[91] 10mm/sec CNT100;
   1:  PR[GP1:91,1] = PR[GP1:90,1] + -71.705;
   1:  PR[GP1:91,2] = PR[GP1:90,2] + 13.559;
   1:L PR[91] 10mm/sec CNT100;
   1:  PR[GP1:91,1] = PR[GP1:90,1] + -72.477;
   1:  PR[GP1:91,2] = PR[GP1:90,2] + 11.322;
   1:L PR[91] 10mm/sec CNT100;
   1:  PR[GP1:91,1] = PR[GP1:90,1] + -72.748;
   1:  PR[GP1:91,2] = PR[GP1:90,2] + 8.878;
   1:L PR[91] 10mm/sec CNT100;
   1:  PR[GP1:91,1] = PR[GP1:90,1] + -74.382;
   1:  PR[GP1:91,2] = PR[GP1:90,2] + 0.256;
   1:L PR[91] 10mm/sec CNT100;
   1:  PR[GP1:91,1] = PR[GP1:90,1] + -74.095;
   1:  PR[GP1:91,2] = PR[GP1:90,2] + -2.320;
   1:L PR[91] 10mm/sec CNT100;
   1:  PR[GP1:91,1] = PR[GP1:90,1] + -72.484;
   1:  PR[GP1:91,2] = PR[GP1:90,2] + -10.742;
   1:L PR[91] 10mm/sec CNT100;
   1:  PR[GP1:91,1] = PR[GP1:90,1] + -71.704;
   1:  PR[GP1:91,2] = PR[GP1:90,2] + -13.004;
   1:L PR[91] 10mm/sec CNT100;
   1:  PR[GP1:91,1] = PR[GP1:90,1] + -70.425;
   1:  PR[GP1:91,2] = PR[GP1:90,2] + -15.074;
   1:L PR[91] 10mm/sec CNT100;
   1:  PR[GP1:91,1] = PR[GP1:90,1] + -65.674;
   1:  PR[GP1:91,2] = PR[GP1:90,2] + -22.573;
   1:L PR[91] 10mm/sec CNT100;
   1:  PR[GP1:91,1] = PR[GP1:90,1] + -64.168;
   1:  PR[GP1:91,2] = PR[GP1:90,2] + -24.111;
   1:L PR[91] 10mm/sec CNT100;
   1:  PR[GP1:91,1] = PR[GP1:90,1] + -62.294;
   1:  PR[GP1:91,2] = PR[GP1:90,2] + -25.323;
   1:L PR[91] 10mm/sec CNT100;
   1:  PR[GP1:91,1] = PR[GP1:90,1] + -54.865;
   1:  PR[GP1:91,2] = PR[GP1:90,2] + -30.756;
   1:L PR[91] 10mm/sec CNT100;
   1:  PR[GP1:91,1] = PR[GP1:90,1] + -53.180;
   1:  PR[GP1:91,2] = PR[GP1:90,2] + -31.377;
   1:L PR[91] 10mm/sec CNT100;
   1:  PR[GP1:91,1] = PR[GP1:90,1] + -43.286;
   1:  PR[GP1:91,2] = PR[GP1:90,2] + -33.943;
   1:L PR[91] 10mm/sec CNT100;
   1:  PR[GP1:91,1] = PR[GP1:90,1] + -42.013;
   1:  PR[GP1:91,2] = PR[GP1:90,2] + -34.111;
   1:L PR[91] 10mm/sec CNT100;
   1:  PR[GP1:91,1] = PR[GP1:90,1] + -40.706;
   1:  PR[GP1:91,2] = PR[GP1:90,2] + -33.993;
   1:L PR[91] 10mm/sec CNT100;
   1:  PR[GP1:91,1] = PR[GP1:90,1] + -29.774;
   1:  PR[GP1:91,2] = PR[GP1:90,2] + -32.674;
   1:L PR[91] 10mm/sec CNT100;
   1:  PR[GP1:91,1] = PR[GP1:90,1] + -29.184;
   1:  PR[GP1:91,2] = PR[GP1:90,2] + -32.484;
   1:L PR[91] 10mm/sec CNT100;
   1:  PR[GP1:91,1] = PR[GP1:90,1] + -28.590;
   1:  PR[GP1:91,2] = PR[GP1:90,2] + -32.134;
   1:L PR[91] 10mm/sec CNT100;
   1:  PR[GP1:91,1] = PR[GP1:90,1] + -18.109;
   1:  PR[GP1:91,2] = PR[GP1:90,2] + -26.511;
   1:L PR[91] 10mm/sec CNT100;
   1:  PR[GP1:91,1] = PR[GP1:90,1] + -17.391;
   1:  PR[GP1:91,2] = PR[GP1:90,2] + -25.660;
   1:L PR[91] 10mm/sec CNT100;
   1:  PR[GP1:91,1] = PR[GP1:90,1] + -9.802;
   1:  PR[GP1:91,2] = PR[GP1:90,2] + -16.861;
   1:L PR[91] 10mm/sec CNT100;
   1:  PR[GP1:91,1] = PR[GP1:90,1] + -9.448;
   1:  PR[GP1:91,2] = PR[GP1:90,2] + -16.099;
   1:L PR[91] 10mm/sec CNT100;
   1:  PR[GP1:91,1] = PR[GP1:90,1] + -5.409;
   1:  PR[GP1:91,2] = PR[GP1:90,2] + -4.433;
   1:L PR[91] 10mm/sec CNT100;
   1:  PR[GP1:91,1] = PR[GP1:90,1] + 4.882;
   1:L PR[91] 10mm/sec CNT100;
   1:  PR[GP1:91,1] = PR[GP1:90,1] + 8.472;
   1:  PR[GP1:91,2] = PR[GP1:90,2] + -15.317;
   1:  PR[GP1:91,3] = PR[GP1:90,3] + 16.775;
   1:L PR[91] 10mm/sec CNT100;
   1:  PR[GP1:91,1] = PR[GP1:90,1] + 9.295;
   1:  PR[GP1:91,2] = PR[GP1:90,2] + -17.090;
   1:L PR[91] 10mm/sec CNT100;
   1:  PR[GP1:91,1] = PR[GP1:90,1] + 16.978;
   1:  PR[GP1:91,2] = PR[GP1:90,2] + -26.004;
   1:L PR[91] 10mm/sec CNT100;
   1:  PR[GP1:91,1] = PR[GP1:90,1] + 17.612;
   1:  PR[GP1:91,2] = PR[GP1:90,2] + -26.625;
   1:L PR[91] 10mm/sec CNT100;
   1:  PR[GP1:91,1] = PR[GP1:90,1] + 25.675;
   1:  PR[GP1:91,2] = PR[GP1:90,2] + -30.860;
   1:L PR[91] 10mm/sec CNT100;
   1:  PR[GP1:91,1] = PR[GP1:90,1] + 28.876;
   1:  PR[GP1:91,2] = PR[GP1:90,2] + -32.586;
   1:L PR[91] 10mm/sec CNT100;
   1:  PR[GP1:91,1] = PR[GP1:90,1] + 28.960;
   1:  PR[GP1:91,2] = PR[GP1:90,2] + -32.613;
   1:L PR[91] 10mm/sec CNT100;
   1:  PR[GP1:91,1] = PR[GP1:90,1] + 41.572;
   1:  PR[GP1:91,2] = PR[GP1:90,2] + -34.111;
   1:L PR[91] 10mm/sec CNT100;
   1:  PR[GP1:91,1] = PR[GP1:90,1] + 42.348;
   1:  PR[GP1:91,2] = PR[GP1:90,2] + -34.008;
   1:L PR[91] 10mm/sec CNT100;
   1:  PR[GP1:91,1] = PR[GP1:90,1] + 53.017;
   1:  PR[GP1:91,2] = PR[GP1:90,2] + -31.242;
   1:L PR[91] 10mm/sec CNT100;
   1:  PR[GP1:91,1] = PR[GP1:90,1] + 54.294;
   1:  PR[GP1:91,2] = PR[GP1:90,2] + -30.772;
   1:L PR[91] 10mm/sec CNT100;
   1:  PR[GP1:91,1] = PR[GP1:90,1] + 55.447;
   1:  PR[GP1:91,2] = PR[GP1:90,2] + -30.025;
   1:L PR[91] 10mm/sec CNT100;
   1:  PR[GP1:91,1] = PR[GP1:90,1] + 63.796;
   1:  PR[GP1:91,2] = PR[GP1:90,2] + -23.949;
   1:L PR[91] 10mm/sec CNT100;
   1:  PR[GP1:91,1] = PR[GP1:90,1] + 65.015;
   1:  PR[GP1:91,2] = PR[GP1:90,2] + -22.704;
   1:L PR[91] 10mm/sec CNT100;
   1:  PR[GP1:91,1] = PR[GP1:90,1] + 65.959;
   1:  PR[GP1:91,2] = PR[GP1:90,2] + -21.177;
   1:L PR[91] 10mm/sec CNT100;
   1:  PR[GP1:91,1] = PR[GP1:90,1] + 71.207;
   1:  PR[GP1:91,2] = PR[GP1:90,2] + -12.890;
   1:L PR[91] 10mm/sec CNT100;
   1:  PR[GP1:91,1] = PR[GP1:90,1] + 71.846;
   1:  PR[GP1:91,2] = PR[GP1:90,2] + -11.038;
   1:L PR[91] 10mm/sec CNT100;
   1:  PR[GP1:91,1] = PR[GP1:90,1] + 72.073;
   1:  PR[GP1:91,2] = PR[GP1:90,2] + -8.997;
   1:L PR[91] 10mm/sec CNT100;
   1:  PR[GP1:91,1] = PR[GP1:90,1] + 73.834;
   1:  PR[GP1:91,2] = PR[GP1:90,2] + 0.302;
   1:L PR[91] 10mm/sec CNT100;
   1:  PR[GP1:91,1] = PR[GP1:90,1] + 73.591;
   1:  PR[GP1:91,2] = PR[GP1:90,2] + 2.491;
   1:L PR[91] 10mm/sec CNT100;
   1:  PR[GP1:91,1] = PR[GP1:90,1] + 71.853;
   1:  PR[GP1:91,2] = PR[GP1:90,2] + 11.573;
   1:L PR[91] 10mm/sec CNT100;
   1:  PR[GP1:91,1] = PR[GP1:90,1] + 71.206;
   1:  PR[GP1:91,2] = PR[GP1:90,2] + 13.452;
   1:L PR[91] 10mm/sec CNT100;
   1:  PR[GP1:91,1] = PR[GP1:90,1] + 70.140;
   1:  PR[GP1:91,2] = PR[GP1:90,2] + 15.176;
   1:L PR[91] 10mm/sec CNT100;
   1:  PR[GP1:91,1] = PR[GP1:90,1] + 65.017;
   1:  PR[GP1:91,2] = PR[GP1:90,2] + 23.260;
   1:L PR[91] 10mm/sec CNT100;
   1:  PR[GP1:91,1] = PR[GP1:90,1] + 63.807;
   1:  PR[GP1:91,2] = PR[GP1:90,2] + 24.495;
   1:L PR[91] 10mm/sec CNT100;
   1:  PR[GP1:91,1] = PR[GP1:90,1] + 62.288;
   1:  PR[GP1:91,2] = PR[GP1:90,2] + 25.478;
   1:L PR[91] 10mm/sec CNT100;
   1:  PR[GP1:91,1] = PR[GP1:90,1] + 54.277;
   1:  PR[GP1:91,2] = PR[GP1:90,2] + 31.336;
   1:L PR[91] 10mm/sec CNT100;
   1:  PR[GP1:91,1] = PR[GP1:90,1] + 53.017;
   1:  PR[GP1:91,2] = PR[GP1:90,2] + 31.800;
   1:L PR[91] 10mm/sec CNT100;
   1:  PR[GP1:91,1] = PR[GP1:90,1] + 42.348;
   1:  PR[GP1:91,2] = PR[GP1:90,2] + 34.566;
   1:L PR[91] 10mm/sec CNT100;
   1:  PR[GP1:91,1] = PR[GP1:90,1] + 41.563;
   1:  PR[GP1:91,2] = PR[GP1:90,2] + 34.670;
   1:L PR[91] 10mm/sec CNT100;
   1:  PR[GP1:91,1] = PR[GP1:90,1] + 40.747;
   1:  PR[GP1:91,2] = PR[GP1:90,2] + 34.596;
   1:L PR[91] 10mm/sec CNT100;
   1:  PR[GP1:91,1] = PR[GP1:90,1] + 28.961;
   1:  PR[GP1:91,2] = PR[GP1:90,2] + 33.171;
   1:L PR[91] 10mm/sec CNT100;
   1:  PR[GP1:91,1] = PR[GP1:90,1] + 28.876;
   1:  PR[GP1:91,2] = PR[GP1:90,2] + 33.144;
   1:L PR[91] 10mm/sec CNT100;
   1:  PR[GP1:91,1] = PR[GP1:90,1] + 25.675;
   1:  PR[GP1:91,2] = PR[GP1:90,2] + 31.418;
   1:L PR[91] 10mm/sec CNT100;
   1:  PR[GP1:91,1] = PR[GP1:90,1] + 17.612;
   1:  PR[GP1:91,2] = PR[GP1:90,2] + 27.183;
   1:L PR[91] 10mm/sec CNT100;
   1:  PR[GP1:91,1] = PR[GP1:90,1] + 16.978;
   1:  PR[GP1:91,2] = PR[GP1:90,2] + 26.562;
   1:L PR[91] 10mm/sec CNT100;
   1:  PR[GP1:91,1] = PR[GP1:90,1] + 9.295;
   1:  PR[GP1:91,2] = PR[GP1:90,2] + 17.648;
   1:L PR[91] 10mm/sec CNT100;
   1:  PR[GP1:91,1] = PR[GP1:90,1] + 8.472;
   1:  PR[GP1:91,2] = PR[GP1:90,2] + 15.874;
   1:L PR[91] 10mm/sec CNT100;
   1:  PR[GP1:91,1] = PR[GP1:90,1] + 4.817;
   1:  PR[GP1:91,2] = PR[GP1:90,2] + 5.316;
   1:L PR[91] 10mm/sec CNT100;
   1:  PR[GP1:91,1] = PR[GP1:90,1] + -5.344;
   1:L PR[91] 10mm/sec CNT100;
   1:  PR[GP1:91,1] = PR[GP1:90,1] + -9.003;
   1:  PR[GP1:91,2] = PR[GP1:90,2] + 15.883;
   1:L PR[91] 10mm/sec CNT100;
   1:  PR[GP1:91,1] = PR[GP1:90,1] + -9.826;
   1:  PR[GP1:91,2] = PR[GP1:90,2] + 17.659;
   1:L PR[91] 10mm/sec CNT100;
   1:  PR[GP1:91,1] = PR[GP1:90,1] + -17.510;
   1:  PR[GP1:91,2] = PR[GP1:90,2] + 26.567;
   1:L PR[91] 10mm/sec CNT100;
   1:  PR[GP1:91,1] = PR[GP1:90,1] + -18.143;
   1:  PR[GP1:91,2] = PR[GP1:90,2] + 27.186;
   1:L PR[91] 10mm/sec CNT100;
   1:  PR[GP1:91,1] = PR[GP1:90,1] + -26.202;
   1:  PR[GP1:91,2] = PR[GP1:90,2] + 31.418;
   1:L PR[91] 10mm/sec CNT100;
   1:  PR[GP1:91,1] = PR[GP1:90,1] + -29.407;
   1:  PR[GP1:91,2] = PR[GP1:90,2] + 33.146;
   1:L PR[91] 10mm/sec CNT100;
   1:  PR[GP1:91,1] = PR[GP1:90,1] + -29.491;
   1:  PR[GP1:91,2] = PR[GP1:90,2] + 33.174;
   1:L PR[91] 10mm/sec CNT100;
   1:  PR[GP1:91,1] = PR[GP1:90,1] + -42.102;
   1:  PR[GP1:91,2] = PR[GP1:90,2] + 34.669;
   1:L PR[91] 10mm/sec CNT100;
   1:  PR[GP1:91,1] = PR[GP1:90,1] + -42.878;
   1:  PR[GP1:91,2] = PR[GP1:90,2] + 34.566;
   1:L PR[91] 10mm/sec CNT100;
   1:  PR[GP1:91,1] = PR[GP1:90,1] + -53.545;
   1:  PR[GP1:91,2] = PR[GP1:90,2] + 31.799;
   1:L PR[91] 10mm/sec CNT100;
   1:  PR[GP1:91,1] = PR[GP1:90,1] + -54.823;
   1:  PR[GP1:91,2] = PR[GP1:90,2] + 31.329;
   1:L PR[91] 10mm/sec CNT100;
   1:  PR[GP1:91,1] = PR[GP1:90,1] + -55.976;
   1:  PR[GP1:91,2] = PR[GP1:90,2] + 30.582;
   1:L PR[91] 10mm/sec CNT100;
   1:  PR[GP1:91,1] = PR[GP1:90,1] + -64.323;
   1:  PR[GP1:91,2] = PR[GP1:90,2] + 24.506;
   1:L PR[91] 10mm/sec CNT100;
   1:  PR[GP1:91,1] = PR[GP1:90,1] + -65.542;
   1:  PR[GP1:91,2] = PR[GP1:90,2] + 23.262;
   1:L PR[91] 10mm/sec CNT100;
   1:  PR[GP1:91,1] = PR[GP1:90,1] + -66.486;
   1:  PR[GP1:91,2] = PR[GP1:90,2] + 21.735;
   1:L PR[91] 10mm/sec CNT100;
   1:  PR[GP1:91,1] = PR[GP1:90,1] + -71.733;
   1:  PR[GP1:91,2] = PR[GP1:90,2] + 13.446;
   1:L PR[91] 10mm/sec CNT100;
   1:  PR[GP1:91,1] = PR[GP1:90,1] + -72.372;
   1:  PR[GP1:91,2] = PR[GP1:90,2] + 11.593;
   1:L PR[91] 10mm/sec CNT100;
   1:  PR[GP1:91,1] = PR[GP1:90,1] + -72.599;
   1:  PR[GP1:91,2] = PR[GP1:90,2] + 9.552;
   1:L PR[91] 10mm/sec CNT100;
   1:  PR[GP1:91,1] = PR[GP1:90,1] + -74.360;
   1:  PR[GP1:91,2] = PR[GP1:90,2] + 0.256;
   1:L PR[91] 10mm/sec CNT100;
   1:  PR[GP1:91,1] = PR[GP1:90,1] + -74.117;
   1:  PR[GP1:91,2] = PR[GP1:90,2] + -1.933;
   1:L PR[91] 10mm/sec CNT100;
   1:  PR[GP1:91,1] = PR[GP1:90,1] + -72.380;
   1:  PR[GP1:91,2] = PR[GP1:90,2] + -11.012;
   1:L PR[91] 10mm/sec CNT100;
   1:  PR[GP1:91,1] = PR[GP1:90,1] + -71.732;
   1:  PR[GP1:91,2] = PR[GP1:90,2] + -12.891;
   1:L PR[91] 10mm/sec CNT100;
   1:  PR[GP1:91,1] = PR[GP1:90,1] + -70.667;
   1:  PR[GP1:91,2] = PR[GP1:90,2] + -14.615;
   1:L PR[91] 10mm/sec CNT100;
   1:  PR[GP1:91,1] = PR[GP1:90,1] + -65.544;
   1:  PR[GP1:91,2] = PR[GP1:90,2] + -22.701;
   1:L PR[91] 10mm/sec CNT100;
   1:  PR[GP1:91,1] = PR[GP1:90,1] + -64.335;
   1:  PR[GP1:91,2] = PR[GP1:90,2] + -23.936;
   1:L PR[91] 10mm/sec CNT100;
   1:  PR[GP1:91,1] = PR[GP1:90,1] + -62.815;
   1:  PR[GP1:91,2] = PR[GP1:90,2] + -24.919;
   1:L PR[91] 10mm/sec CNT100;
   1:  PR[GP1:91,1] = PR[GP1:90,1] + -54.806;
   1:  PR[GP1:91,2] = PR[GP1:90,2] + -30.777;
   1:L PR[91] 10mm/sec CNT100;
   1:  PR[GP1:91,1] = PR[GP1:90,1] + -53.545;
   1:  PR[GP1:91,2] = PR[GP1:90,2] + -31.241;
   1:L PR[91] 10mm/sec CNT100;
   1:  PR[GP1:91,1] = PR[GP1:90,1] + -42.878;
   1:  PR[GP1:91,2] = PR[GP1:90,2] + -34.008;
   1:L PR[91] 10mm/sec CNT100;
   1:  PR[GP1:91,1] = PR[GP1:90,1] + -42.093;
   1:  PR[GP1:91,2] = PR[GP1:90,2] + -34.112;
   1:L PR[91] 10mm/sec CNT100;
   1:  PR[GP1:91,1] = PR[GP1:90,1] + -41.277;
   1:  PR[GP1:91,2] = PR[GP1:90,2] + -34.038;
   1:L PR[91] 10mm/sec CNT100;
   1:  PR[GP1:91,1] = PR[GP1:90,1] + -29.492;
   1:  PR[GP1:91,2] = PR[GP1:90,2] + -32.616;
   1:L PR[91] 10mm/sec CNT100;
   1:  PR[GP1:91,1] = PR[GP1:90,1] + -29.407;
   1:  PR[GP1:91,2] = PR[GP1:90,2] + -32.588;
   1:L PR[91] 10mm/sec CNT100;
   1:  PR[GP1:91,1] = PR[GP1:90,1] + -26.202;
   1:  PR[GP1:91,2] = PR[GP1:90,2] + -30.859;
   1:L PR[91] 10mm/sec CNT100;
   1:  PR[GP1:91,1] = PR[GP1:90,1] + -18.143;
   1:  PR[GP1:91,2] = PR[GP1:90,2] + -26.628;
   1:L PR[91] 10mm/sec CNT100;
   1:  PR[GP1:91,1] = PR[GP1:90,1] + -17.510;
   1:  PR[GP1:91,2] = PR[GP1:90,2] + -26.009;
   1:L PR[91] 10mm/sec CNT100;
   1:  PR[GP1:91,1] = PR[GP1:90,1] + -9.826;
   1:  PR[GP1:91,2] = PR[GP1:90,2] + -17.101;
   1:L PR[91] 10mm/sec CNT100;
   1:  PR[GP1:91,1] = PR[GP1:90,1] + -9.002;
   1:  PR[GP1:91,2] = PR[GP1:90,2] + -15.324;
   1:L PR[91] 10mm/sec CNT100;
   1:  PR[GP1:91,1] = PR[GP1:90,1] + -5.344;
   1:  PR[GP1:91,2] = PR[GP1:90,2] + -4.758;
   1:L PR[91] 10mm/sec CNT100;
   1:  PR[GP1:91,1] = PR[GP1:90,1] + 4.817;
   1:L PR[91] 10mm/sec CNT100;
   1:  PR[GP1:91,1] = PR[GP1:90,1] + 8.026;
   1:  PR[GP1:91,2] = PR[GP1:90,2] + -14.543;
   1:  PR[GP1:91,3] = PR[GP1:90,3] + 17.385;
   1:L PR[91] 10mm/sec CNT100;
   1:  PR[GP1:91,1] = PR[GP1:90,1] + 9.320;
   1:  PR[GP1:91,2] = PR[GP1:90,2] + -17.329;
   1:L PR[91] 10mm/sec CNT100;
   1:  PR[GP1:91,1] = PR[GP1:90,1] + 16.258;
   1:  PR[GP1:91,2] = PR[GP1:90,2] + -25.380;
   1:L PR[91] 10mm/sec CNT100;
   1:  PR[GP1:91,1] = PR[GP1:90,1] + 17.675;
   1:  PR[GP1:91,2] = PR[GP1:90,2] + -26.768;
   1:L PR[91] 10mm/sec CNT100;
   1:  PR[GP1:91,1] = PR[GP1:90,1] + 28.429;
   1:  PR[GP1:91,2] = PR[GP1:90,2] + -32.415;
   1:L PR[91] 10mm/sec CNT100;
   1:  PR[GP1:91,1] = PR[GP1:90,1] + 28.923;
   1:  PR[GP1:91,2] = PR[GP1:90,2] + -32.632;
   1:L PR[91] 10mm/sec CNT100;
   1:  PR[GP1:91,1] = PR[GP1:90,1] + 34.449;
   1:  PR[GP1:91,2] = PR[GP1:90,2] + -33.252;
   1:L PR[91] 10mm/sec CNT100;
   1:  PR[GP1:91,1] = PR[GP1:90,1] + 41.652;
   1:  PR[GP1:91,2] = PR[GP1:90,2] + -34.111;
   1:L PR[91] 10mm/sec CNT100;
   1:  PR[GP1:91,1] = PR[GP1:90,1] + 41.940;
   1:  PR[GP1:91,2] = PR[GP1:90,2] + -34.073;
   1:L PR[91] 10mm/sec CNT100;
   1:  PR[GP1:91,1] = PR[GP1:90,1] + 53.382;
   1:  PR[GP1:91,2] = PR[GP1:90,2] + -31.106;
   1:L PR[91] 10mm/sec CNT100;
   1:  PR[GP1:91,1] = PR[GP1:90,1] + 54.235;
   1:  PR[GP1:91,2] = PR[GP1:90,2] + -30.792;
   1:L PR[91] 10mm/sec CNT100;
   1:  PR[GP1:91,1] = PR[GP1:90,1] + 55.009;
   1:  PR[GP1:91,2] = PR[GP1:90,2] + -30.291;
   1:L PR[91] 10mm/sec CNT100;
   1:  PR[GP1:91,1] = PR[GP1:90,1] + 63.962;
   1:  PR[GP1:91,2] = PR[GP1:90,2] + -23.774;
   1:L PR[91] 10mm/sec CNT100;
   1:  PR[GP1:91,1] = PR[GP1:90,1] + 64.885;
   1:  PR[GP1:91,2] = PR[GP1:90,2] + -22.832;
   1:L PR[91] 10mm/sec CNT100;
   1:  PR[GP1:91,1] = PR[GP1:90,1] + 65.606;
   1:  PR[GP1:91,2] = PR[GP1:90,2] + -21.665;
   1:L PR[91] 10mm/sec CNT100;
   1:  PR[GP1:91,1] = PR[GP1:90,1] + 71.235;
   1:  PR[GP1:91,2] = PR[GP1:90,2] + -12.777;
   1:L PR[91] 10mm/sec CNT100;
   1:  PR[GP1:91,1] = PR[GP1:90,1] + 71.742;
   1:  PR[GP1:91,2] = PR[GP1:90,2] + -11.308;
   1:L PR[91] 10mm/sec CNT100;
   1:  PR[GP1:91,1] = PR[GP1:90,1] + 71.924;
   1:  PR[GP1:91,2] = PR[GP1:90,2] + -9.672;
   1:L PR[91] 10mm/sec CNT100;
   1:  PR[GP1:91,1] = PR[GP1:90,1] + 73.813;
   1:  PR[GP1:91,2] = PR[GP1:90,2] + 0.302;
   1:L PR[91] 10mm/sec CNT100;
   1:  PR[GP1:91,1] = PR[GP1:90,1] + 73.612;
   1:  PR[GP1:91,2] = PR[GP1:90,2] + 2.103;
   1:L PR[91] 10mm/sec CNT100;
   1:  PR[GP1:91,1] = PR[GP1:90,1] + 71.749;
   1:  PR[GP1:91,2] = PR[GP1:90,2] + 11.844;
   1:L PR[91] 10mm/sec CNT100;
   1:  PR[GP1:91,1] = PR[GP1:90,1] + 71.234;
   1:  PR[GP1:91,2] = PR[GP1:90,2] + 13.339;
   1:L PR[91] 10mm/sec CNT100;
   1:  PR[GP1:91,1] = PR[GP1:90,1] + 70.382;
   1:  PR[GP1:91,2] = PR[GP1:90,2] + 14.717;
   1:L PR[91] 10mm/sec CNT100;
   1:  PR[GP1:91,1] = PR[GP1:90,1] + 64.887;
   1:  PR[GP1:91,2] = PR[GP1:90,2] + 23.388;
   1:L PR[91] 10mm/sec CNT100;
   1:  PR[GP1:91,1] = PR[GP1:90,1] + 63.974;
   1:  PR[GP1:91,2] = PR[GP1:90,2] + 24.321;
   1:L PR[91] 10mm/sec CNT100;
   1:  PR[GP1:91,1] = PR[GP1:90,1] + 62.810;
   1:  PR[GP1:91,2] = PR[GP1:90,2] + 25.074;
   1:L PR[91] 10mm/sec CNT100;
   1:  PR[GP1:91,1] = PR[GP1:90,1] + 54.218;
   1:  PR[GP1:91,2] = PR[GP1:90,2] + 31.356;
   1:L PR[91] 10mm/sec CNT100;
   1:  PR[GP1:91,1] = PR[GP1:90,1] + 53.382;
   1:  PR[GP1:91,2] = PR[GP1:90,2] + 31.664;
   1:L PR[91] 10mm/sec CNT100;
   1:  PR[GP1:91,1] = PR[GP1:90,1] + 41.940;
   1:  PR[GP1:91,2] = PR[GP1:90,2] + 34.631;
   1:L PR[91] 10mm/sec CNT100;
   1:  PR[GP1:91,1] = PR[GP1:90,1] + 41.644;
   1:  PR[GP1:91,2] = PR[GP1:90,2] + 34.670;
   1:L PR[91] 10mm/sec CNT100;
   1:  PR[GP1:91,1] = PR[GP1:90,1] + 41.318;
   1:  PR[GP1:91,2] = PR[GP1:90,2] + 34.641;
   1:L PR[91] 10mm/sec CNT100;
   1:  PR[GP1:91,1] = PR[GP1:90,1] + 34.449;
   1:  PR[GP1:91,2] = PR[GP1:90,2] + 33.810;
   1:L PR[91] 10mm/sec CNT100;
   1:  PR[GP1:91,1] = PR[GP1:90,1] + 28.923;
   1:  PR[GP1:91,2] = PR[GP1:90,2] + 33.190;
   1:L PR[91] 10mm/sec CNT100;
   1:  PR[GP1:91,1] = PR[GP1:90,1] + 28.429;
   1:  PR[GP1:91,2] = PR[GP1:90,2] + 32.973;
   1:L PR[91] 10mm/sec CNT100;
   1:  PR[GP1:91,1] = PR[GP1:90,1] + 17.675;
   1:  PR[GP1:91,2] = PR[GP1:90,2] + 27.326;
   1:L PR[91] 10mm/sec CNT100;
   1:  PR[GP1:91,1] = PR[GP1:90,1] + 16.258;
   1:  PR[GP1:91,2] = PR[GP1:90,2] + 25.937;
   1:L PR[91] 10mm/sec CNT100;
   1:  PR[GP1:91,1] = PR[GP1:90,1] + 9.320;
   1:  PR[GP1:91,2] = PR[GP1:90,2] + 17.887;
   1:L PR[91] 10mm/sec CNT100;
   1:  PR[GP1:91,1] = PR[GP1:90,1] + 8.026;
   1:  PR[GP1:91,2] = PR[GP1:90,2] + 15.099;
   1:L PR[91] 10mm/sec CNT100;
   1:  PR[GP1:91,1] = PR[GP1:90,1] + 4.751;
   1:  PR[GP1:91,2] = PR[GP1:90,2] + 5.641;
   1:L PR[91] 10mm/sec CNT100;
   1:  PR[GP1:91,1] = PR[GP1:90,1] + -5.279;
   1:L PR[91] 10mm/sec CNT100;
   1:  PR[GP1:91,1] = PR[GP1:90,1] + -8.557;
   1:  PR[GP1:91,2] = PR[GP1:90,2] + 15.108;
   1:L PR[91] 10mm/sec CNT100;
   1:  PR[GP1:91,1] = PR[GP1:90,1] + -9.851;
   1:  PR[GP1:91,2] = PR[GP1:90,2] + 17.899;
   1:L PR[91] 10mm/sec CNT100;
   1:  PR[GP1:91,1] = PR[GP1:90,1] + -16.790;
   1:  PR[GP1:91,2] = PR[GP1:90,2] + 25.944;
   1:L PR[91] 10mm/sec CNT100;
   1:  PR[GP1:91,1] = PR[GP1:90,1] + -18.207;
   1:  PR[GP1:91,2] = PR[GP1:90,2] + 27.329;
   1:L PR[91] 10mm/sec CNT100;
   1:  PR[GP1:91,1] = PR[GP1:90,1] + -28.961;
   1:  PR[GP1:91,2] = PR[GP1:90,2] + 32.976;
   1:L PR[91] 10mm/sec CNT100;
   1:  PR[GP1:91,1] = PR[GP1:90,1] + -29.454;
   1:  PR[GP1:91,2] = PR[GP1:90,2] + 33.192;
   1:L PR[91] 10mm/sec CNT100;
   1:  PR[GP1:91,1] = PR[GP1:90,1] + -34.975;
   1:  PR[GP1:91,2] = PR[GP1:90,2] + 33.811;
   1:L PR[91] 10mm/sec CNT100;
   1:  PR[GP1:91,1] = PR[GP1:90,1] + -42.183;
   1:  PR[GP1:91,2] = PR[GP1:90,2] + 34.669;
   1:L PR[91] 10mm/sec CNT100;
   1:  PR[GP1:91,1] = PR[GP1:90,1] + -42.471;
   1:  PR[GP1:91,2] = PR[GP1:90,2] + 34.631;
   1:L PR[91] 10mm/sec CNT100;
   1:  PR[GP1:91,1] = PR[GP1:90,1] + -53.911;
   1:  PR[GP1:91,2] = PR[GP1:90,2] + 31.663;
   1:L PR[91] 10mm/sec CNT100;
   1:  PR[GP1:91,1] = PR[GP1:90,1] + -54.764;
   1:  PR[GP1:91,2] = PR[GP1:90,2] + 31.349;
   1:L PR[91] 10mm/sec CNT100;
   1:  PR[GP1:91,1] = PR[GP1:90,1] + -55.538;
   1:  PR[GP1:91,2] = PR[GP1:90,2] + 30.848;
   1:L PR[91] 10mm/sec CNT100;
   1:  PR[GP1:91,1] = PR[GP1:90,1] + -64.489;
   1:  PR[GP1:91,2] = PR[GP1:90,2] + 24.332;
   1:L PR[91] 10mm/sec CNT100;
   1:  PR[GP1:91,1] = PR[GP1:90,1] + -65.412;
   1:  PR[GP1:91,2] = PR[GP1:90,2] + 23.390;
   1:L PR[91] 10mm/sec CNT100;
   1:  PR[GP1:91,1] = PR[GP1:90,1] + -66.134;
   1:  PR[GP1:91,2] = PR[GP1:90,2] + 22.222;
   1:L PR[91] 10mm/sec CNT100;
   1:  PR[GP1:91,1] = PR[GP1:90,1] + -71.761;
   1:  PR[GP1:91,2] = PR[GP1:90,2] + 13.333;
   1:L PR[91] 10mm/sec CNT100;
   1:  PR[GP1:91,1] = PR[GP1:90,1] + -72.268;
   1:  PR[GP1:91,2] = PR[GP1:90,2] + 11.864;
   1:L PR[91] 10mm/sec CNT100;
   1:  PR[GP1:91,1] = PR[GP1:90,1] + -72.450;
   1:  PR[GP1:91,2] = PR[GP1:90,2] + 10.227;
   1:L PR[91] 10mm/sec CNT100;
